// TwinCAT 3 PLC project WidgetSample
// ProgramVersion: 3.1.4026.20
// libraries:
//   Tc2_Standard, * (Beckhoff Automation GmbH)
//   Tc2_System, * (Beckhoff Automation GmbH)
//   Tc3_IotCommunicator, * (Beckhoff Automation GmbH)
//   Tc3_Module, * (Beckhoff Automation GmbH)
// project tree:
//   DUTs/4ChannelLED/ ST_Widgets_RGBWEL2564.TcDUT, ST_Widget_RGBWEL2564_Template.TcDUT
//   DUTs/AC/ ST_Widgets_AC.TcDUT, ST_Widget_AC_AlternativeTemplate.TcDUT, ST_Widget_AC_Template.TcDUT
//   DUTs/BarChart/ ST_Widgets_BarChart.TcDUT, ST_Widget_BarChart_Template.TcDUT
//   DUTs/Blinds/ ST_Widgets_Blinds.TcDUT, ST_Widget_SimpleBlinds_Template.TcDUT, ST_Widget_Blinds_Template.TcDUT
//   DUTs/ChargingStation/ ST_Widgets_ChargingStations.TcDUT, ST_Widget_ChargingStation_Template.TcDUT
//   DUTs/EnergyMonitoring/ ST_Widgets_EnergyMonitoring.TcDUT, ST_Widget_EnergyMonitoring_Template.TcDUT
//   DUTs/GeneralWidget/ ST_Widgets_GeneralWidget.TcDUT, ST_Widget_GeneralWidget_AlternativeTemplate.TcDUT, ST_Widget_GeneralWidget_Template.TcDUT
//   DUTs/Lighting/ ST_Widgets_Lightings.TcDUT, ST_Widget_Lighting_Template.TcDUT
//   DUTs/Plugs/ ST_Widgets_Plugs.TcDUT, ST_Widget_Plug_Template.TcDUT
//   DUTs/RGBW/ ST_Widgets_RGBW.TcDUT, ST_Widget_RGBW_Template.TcDUT
//   DUTs/ ST_JsonData.TcDUT, ST_WidgetData.TcDUT, ST_Widgets_Overview.TcDUT
//   DUTs/TimeSwitch/ ST_Widgets_TimeSwitch.TcDUT, ST_Widget_TimeSwitch_Template.TcDUT
//   DUTs/Ventilation/ ST_Widgets_Ventilation.TcDUT, ST_Widget_Ventilation_AlternativeTemplate.TcDUT, ST_Widget_Ventilation_Template.TcDUT
//   GVLs/ GVL_Widgets.TcGVL
//   / PlcTask.TcTTO
//   POUs/ MAIN.TcPOU, WidgetValues.TcPOU
// real-time tasks:
//   TASK PlcTask: cycle T#10ms, priority 20, ADS port 350

CONFIGURATION WidgetSample
    RESOURCE PLC ON TwinCAT3
        TASK PlcTask(INTERVAL := T#10ms, PRIORITY := 20);
        PROGRAM MAIN WITH PlcTask : MAIN;
    END_RESOURCE
END_CONFIGURATION

// ---- DUTs/4ChannelLED/ST_Widgets_RGBWEL2564.TcDUT
TYPE ST_Widgets_RGBWEL2564 :
STRUCT
	{attribute 'iot.ReadOnly' := 'true'}
	{attribute 'iot.DisplayName' := ' RGBW EL2564 Sample 1'}
	{attribute 'iot.WidgetType' := 'RGBWEL2564'}
	{attribute 'iot.LedRedSliderVisible' := 'true'}
	{attribute 'iot.LedGreenSliderVisible' := 'true'}
	{attribute 'iot.LedBlueSliderVisible' := 'true'}
	{attribute 'iot.LedWhiteSliderVisible' := 'true'}
	{attribute 'iot.LedModeVisible' := 'false'}
	{attribute 'iot.LedModeChangeable' := 'false'}
	stRGBWLed1	: ST_Widget_RGBWEL2564_Template;
	
	{attribute 'iot.ReadOnly' := 'false'}
	{attribute 'iot.DisplayName' := 'RGBW EL2564 Sample 2'}
	{attribute 'iot.WidgetType' := 'RGBWEL2564'}
	{attribute 'iot.LedRedSliderVisible' := 'true'}
	{attribute 'iot.LedGreenSliderVisible' := 'true'}
	{attribute 'iot.LedBlueSliderVisible' := 'true'}
	{attribute 'iot.LedWhiteSliderVisible' := 'true'}
	{attribute 'iot.LedModeVisible' := 'true'}
	{attribute 'iot.LedModeChangeable' := 'true'}
	stRGBWLed2	: ST_Widget_RGBWEL2564_Template;
	
	{attribute 'iot.ReadOnly' := 'false'}
	{attribute 'iot.DisplayName' := 'RGBW EL2564 Sample 3'}
	{attribute 'iot.WidgetType' := 'RGBWEL2564'}
	{attribute 'iot.LedRedSliderVisible' := 'true'}
	{attribute 'iot.LedGreenSliderVisible' := 'true'}
	{attribute 'iot.LedBlueSliderVisible' := 'true'}
	{attribute 'iot.LedWhiteSliderVisible' := 'true'}
	{attribute 'iot.LedModeVisible' := 'true'}
	{attribute 'iot.LedModeChangeable' := 'true'}
	stRGBWLed3	: ST_Widget_RGBWEL2564_Template;
END_STRUCT
END_TYPE

// ---- DUTs/4ChannelLED/ST_Widget_RGBWEL2564_Template.TcDUT
TYPE ST_Widget_RGBWEL2564_Template :
STRUCT
	sDisplayName	: STRING := ''; // Insert STRING here to overwrite iot.DisplayName

	bOn				: BOOL;
	
	nRed			: INT;
	nGreen			: INT;
	nBlue			: INT;
	nWhite			: INT;

	sMode			: STRING; // can be set to any value, does not have to match the array below
	aModes			: ARRAY[0..1] OF STRING;
END_STRUCT
END_TYPE

// ---- DUTs/AC/ST_Widgets_AC.TcDUT
TYPE ST_Widgets_AC :
STRUCT
	{attribute 'iot.ReadOnly' := 'false'}
	{attribute 'iot.DisplayName' := 'AC Sample 1'}
	{attribute 'iot.WidgetType' := 'AC'}
	{attribute 'iot.ACValueRequestVisible' := 'true'}
	{attribute 'iot.ACSliderVisible' := 'false'}
	{attribute 'iot.ACModeVisible' := 'false'}
	{attribute 'iot.ACModeChangeable' := 'false'}
	{attribute 'iot.ACModeStrengthVisible' := 'true'}
	{attribute 'iot.ACModeStrengthChangeable' := 'true'}
	{attribute 'iot.ACModeLamellaVisible' := 'true'}
	{attribute 'iot.ACModeLamellaChangeable' := 'true'}
	stAC1			: ST_Widget_AC_AlternativeTemplate;
	
	{attribute 'iot.ReadOnly' := 'false'}
	{attribute 'iot.DisplayName' := 'AC Sample 2'}
	{attribute 'iot.WidgetType' := 'AC'}
	{attribute 'iot.ACValueRequestVisible' := 'true'}
	{attribute 'iot.ACSliderVisible' := 'true'}
	{attribute 'iot.ACModeVisible' := 'true'}
	{attribute 'iot.ACModeChangeable' := 'true'}
	{attribute 'iot.ACModeStrengthVisible' := 'true'}
	{attribute 'iot.ACModeStrengthChangeable' := 'true'}
	{attribute 'iot.ACModeLamellaVisible' := 'true'}
	{attribute 'iot.ACModeLamellaChangeable' := 'true'}
	stAC2			: ST_Widget_AC_Template;
	
	{attribute 'iot.ReadOnly' := 'true'}
	{attribute 'iot.DisplayName' := 'AC Sample 3'}
	{attribute 'iot.WidgetType' := 'AC'}
	{attribute 'iot.ACValueRequestVisible' := 'false'}
	{attribute 'iot.ACSliderVisible' := 'true'}
	{attribute 'iot.ACModeVisible' := 'true'}
	{attribute 'iot.ACModeChangeable' := 'false'}
	{attribute 'iot.ACModeStrengthVisible' := 'true'}
	{attribute 'iot.ACModeStrengthChangeable' := 'false'}
	{attribute 'iot.ACModeLamellaVisible' := 'false'}
	{attribute 'iot.ACModeLamellaChangeable' := 'false'}
	stAC3			: ST_Widget_AC_Template;
END_STRUCT
END_TYPE

// ---- DUTs/AC/ST_Widget_AC_AlternativeTemplate.TcDUT
TYPE ST_Widget_AC_AlternativeTemplate :
STRUCT
	sDisplayName	: STRING := ''; // Insert STRING here to overwrite iot.DisplayName

	nAcMode			: INT;	// 0: Off, 1: Cooling, 2: Ventilating, 3: Heating, 4: Cooling Off, 5: Ventilating Off, 6: Heating Off
	
	{attribute 'iot.Unit':='°F'}
	{attribute 'iot.MinValue':='64'}
	{attribute 'iot.MaxValue':='73'}
	nTemperature		: LREAL;	
	nTemperatureRequest : LREAL;
	
	sMode			: STRING; // can be set to any value, does not have to match the array below
	aModes			: ARRAY[0..2] OF STRING;
	sMode_Strength	: STRING;
	aModes_Strength	: ARRAY[0..2] OF STRING;
	sMode_Lamella	: STRING;
	aModes_Lamella	: ARRAY[0..1] OF STRING;
END_STRUCT
END_TYPE

// ---- DUTs/AC/ST_Widget_AC_Template.TcDUT
TYPE ST_Widget_AC_Template :
STRUCT
	sDisplayName	: STRING := ''; // Insert STRING here to overwrite iot.DisplayName

	nAcMode			: INT;	// 0: Off, 1: Cooling, 2: Ventilating, 3: Heating, 4: Cooling Off, 5: Ventilating Off, 6: Heating Off
	
	{attribute 'iot.Unit':='°C'}
	{attribute 'iot.MinValue':='18'}
	{attribute 'iot.MaxValue':='23'}
	nTemperature		: LREAL;	
	nTemperatureRequest : LREAL;
	
	sMode			: STRING; // can be set to any value, does not have to match the array below
	aModes			: ARRAY[0..2] OF STRING;
	sMode_Strength	: STRING;
	aModes_Strength	: ARRAY[0..2] OF STRING;
	sMode_Lamella	: STRING;
	aModes_Lamella	: ARRAY[0..1] OF STRING;
END_STRUCT
END_TYPE

// ---- DUTs/BarChart/ST_Widgets_BarChart.TcDUT
TYPE ST_Widgets_BarChart :
STRUCT
	{attribute 'iot.DisplayName' := 'Chart Widget'}
	{attribute 'iot.WidgetType' := 'BarChart'}
	{attribute 'iot.ChartXAxisLabel' := 'Power consumption'}
	{attribute 'iot.ChartYAxisLabel' := 'Weekdays'}
	{attribute 'iot.Unit' := 'kW/h'}
	{attribute 'iot.ChartLegendVisible' := 'true'}
	{attribute 'iot.ChartValuesVisible' := 'true'}
	{attribute 'iot.MinValue':='0'}
	{attribute 'iot.MaxValue':='1550'}
	{attribute 'iot.ChartBarColor1' := '#FF80AC'}
	{attribute 'iot.ChartBarColor2' := '#FF00FF'}
	stBarChart1	: St_Widget_BarChart_Template;
	
	{attribute 'iot.DisplayName' := 'Chart Widget'}
	{attribute 'iot.WidgetType' := 'BarChart'}
	{attribute 'iot.ChartXAxisLabel' := 'Power consumption'}
	{attribute 'iot.ChartYAxisLabel' := 'Weekdays'}
	{attribute 'iot.Unit' := 'kW/h'}
	{attribute 'iot.ChartLegendVisible' := 'true'}
	{attribute 'iot.ChartValuesVisible' := 'true'}
	{attribute 'iot.MinValue':='0'}
	{attribute 'iot.MaxValue':='1600'}
	{attribute 'iot.ChartBarColor1' := '#00FFFF'}
	{attribute 'iot.ChartBarColor2' := '#0091AA'}
	stBarChart2	: St_Widget_BarChart_Template;
END_STRUCT
END_TYPE

// ---- DUTs/BarChart/ST_Widget_BarChart_Template.TcDUT
TYPE ST_Widget_BarChart_Template :
STRUCT
	sDisplayName	: STRING := '';

	aDataSeries			: ARRAY[0..6] OF INT;
	aComparismDataSeries: ARRAY[0..6] OF INT;
	aDataSeriesIdentifier:ARRAY[0..6] OF STRING;
	
	aLegendLabels		: ARRAY[0..1] OF STRING;
END_STRUCT
END_TYPE

// ---- DUTs/Blinds/ST_Widgets_Blinds.TcDUT
TYPE ST_Widgets_Blinds :
STRUCT
	{attribute 'iot.ReadOnly' := 'true'}
	{attribute 'iot.DisplayName' := 'Blinds Sample 1'}
	{attribute 'iot.WidgetType' := 'Blinds'}
	{attribute 'iot.BlindsPositionValueVisible' := 'true'}
	{attribute 'iot.BlindsPositionSliderVisible' := 'true'}
	{attribute 'iot.BlindsAngleValueVisible' := 'false'} 
	{attribute 'iot.BlindsAngleSliderVisible' := 'false'}
	{attribute 'iot.BlindsModeVisible' := 'true'} 
	{attribute 'iot.BlindsModeChangeable' := 'false'}
	stBlinds1	: ST_Widget_Blinds_Template;
	
	{attribute 'iot.ReadOnly' := 'false'}
	{attribute 'iot.DisplayName' := 'Blinds Sample 2'}
	{attribute 'iot.WidgetType' := 'Blinds'}
	{attribute 'iot.BlindsPositionValueVisible' := 'true'}
	{attribute 'iot.BlindsPositionSliderVisible' := 'true'}
	{attribute 'iot.BlindsAngleValueVisible' := 'false'} 
	{attribute 'iot.BlindsAngleSliderVisible' := 'false'}
	{attribute 'iot.BlindsModeVisible' := 'false'} 
	{attribute 'iot.BlindsModeChangeable' := 'false'}
	stBlinds2	: ST_Widget_Blinds_Template;
	
	{attribute 'iot.ReadOnly' := 'false'}
	{attribute 'iot.DisplayName' := 'Blinds Sample 3'}
	{attribute 'iot.WidgetType' := 'Blinds'}
	{attribute 'iot.BlindsPositionValueVisible' := 'true'}
	{attribute 'iot.BlindsPositionSliderVisible' := 'true'}
	{attribute 'iot.BlindsAngleValueVisible' := 'true'} 
	{attribute 'iot.BlindsAngleSliderVisible' := 'true'}
	{attribute 'iot.BlindsModeVisible' := 'true'} 
	{attribute 'iot.BlindsModeChangeable' := 'true'}
	stBlinds3	: ST_Widget_Blinds_Template;
	
	{attribute 'iot.ReadOnly' := 'false'}
	{attribute 'iot.DisplayName' := 'Simple Blinds Sample 1'}
	{attribute 'iot.WidgetType' := 'SimpleBlinds'}
	{attribute 'iot.BlindsPositionSliderVisible' := 'true'}
	stSimpleBlinds1	: ST_Widget_SimpleBlinds_Template;
	
	{attribute 'iot.ReadOnly' := 'false'}
	{attribute 'iot.DisplayName' := 'Simple Blinds Sample 2'}
	{attribute 'iot.WidgetType' := 'SimpleBlinds'}
	{attribute 'iot.BlindsPositionSliderVisible' := 'false'}
	stSimpleBlinds2	: ST_Widget_SimpleBlinds_Template;
END_STRUCT
END_TYPE

// ---- DUTs/Blinds/ST_Widget_SimpleBlinds_Template.TcDUT
TYPE ST_Widget_SimpleBlinds_Template :
STRUCT
	sDisplayName		: STRING := ''; // Insert STRING here to overwrite iot.DisplayName
	
	bPositionUp			: BOOL;
	bPositionDown		: BOOL;
	{attribute 'iot.MinValue':='0'}
	{attribute 'iot.MaxValue':='100'}
	nPositionValue		: INT;
END_STRUCT
END_TYPE

// ---- DUTs/Blinds/ST_Widget_Blinds_Template.TcDUT
TYPE ST_Widget_Blinds_Template :
STRUCT
	sDisplayName		: STRING := ''; // Insert STRING here to overwrite iot.DisplayName
	bActive				: BOOL;
	bPositionUp			: BOOL;
	bPositionDown		: BOOL;
	bAngleUp			: BOOL;
	bAngleDown			: BOOL;
	{attribute 'iot.Unit':='%'}
	{attribute 'iot.MinValue':='0'}
	{attribute 'iot.MaxValue':='100'}
	nPositionValue		: INT;	
	nPositionRequest 	: INT;
	{attribute 'iot.Unit':='°'}
	{attribute 'iot.MinValue':='-90'}
	{attribute 'iot.MaxValue':='90'}
	nAngleValue			: INT;
	nAngleRequest 		: INT;	
	sMode				: STRING; // can be set to any value, does not have to match the array below
	aModes				: ARRAY[0..1] OF STRING;
END_STRUCT
END_TYPE

// ---- DUTs/ChargingStation/ST_Widgets_ChargingStations.TcDUT
TYPE ST_Widgets_ChargingStations :
STRUCT
	{attribute 'iot.ReadOnly' := 'false'}
	{attribute 'iot.DisplayName' := 'Charging Station Sample 1'}
	{attribute 'iot.WidgetType' := 'ChargingStation'}
	{attribute 'iot.ChargingStationReserveVisible' := 'true'} 
	{attribute 'iot.ChargingStationPhase2Visible' := 'true'} 
	{attribute 'iot.ChargingStationPhase3Visible' := 'true'} 
	stChargingStation1	: ST_Widget_ChargingStation_Template;
	
	{attribute 'iot.ReadOnly' := 'false'}
	{attribute 'iot.DisplayName' := 'Charging Station Sample 2'}
	{attribute 'iot.WidgetType' := 'ChargingStation'}
	{attribute 'iot.ChargingStationReserveVisible' := 'false'} 
	{attribute 'iot.ChargingStationPhase2Visible' := 'true'} 
	{attribute 'iot.ChargingStationPhase3Visible' := 'false'} 
	stChargingStation2	: ST_Widget_ChargingStation_Template;
END_STRUCT
END_TYPE

// ---- DUTs/ChargingStation/ST_Widget_ChargingStation_Template.TcDUT
TYPE ST_Widget_ChargingStation_Template :
STRUCT
	sDisplayName				: STRING;
	
	bStartCharging				: BOOL;
	bStopCharging				: BOOL;
	bReserveCharging			: BOOL;
	
	sStatus						: STRING;	
	nBatteryLevel				: UINT;
	nCurrentPower				: LREAL;
	aThreePhaseMaxPower			: ARRAY[0..2] OF LREAL;
	aThreePhaseCurrentPower		: ARRAY[0..2] OF LREAL;
	aThreePhaseAmperage			: ARRAY[0..2] OF LREAL;
	aThreePhaseVoltage			: ARRAY[0..2] OF LREAL;
	nChargingTime				: UDINT;
	nChargingEnergy				: LREAL;
END_STRUCT
END_TYPE

// ---- DUTs/EnergyMonitoring/ST_Widgets_EnergyMonitoring.TcDUT
TYPE ST_Widgets_EnergyMonitoring :
STRUCT
	{attribute 'iot.ReadOnly' := 'false'}
	{attribute 'iot.DisplayName' := 'Energy Monitoring Sample 1'}
	{attribute 'iot.WidgetType' := 'EnergyMonitoring'}
	{attribute 'iot.EnergyMonitoringPhase2Visible' := 'true'} 
	{attribute 'iot.EnergyMonitoringPhase3Visible' := 'true'} 
	stEnergyMonitoring1	: ST_Widget_EnergyMonitoring_Template;
	
	{attribute 'iot.ReadOnly' := 'false'}
	{attribute 'iot.DisplayName' := 'Energy Monitoring Sample 2'}
	{attribute 'iot.WidgetType' := 'EnergyMonitoring'}
	{attribute 'iot.EnergyMonitoringPhase2Visible' := 'true'} 
	{attribute 'iot.EnergyMonitoringPhase3Visible' := 'false'} 
	stEnergyMonitoring2	: ST_Widget_EnergyMonitoring_Template;
	
	{attribute 'iot.ReadOnly' := 'false'}
	{attribute 'iot.DisplayName' := 'Energy Monitoring Sample 3'}
	{attribute 'iot.WidgetType' := 'EnergyMonitoring'}
	{attribute 'iot.EnergyMonitoringPhase2Visible' := 'false'} 
	{attribute 'iot.EnergyMonitoringPhase3Visible' := 'false'} 
	stEnergyMonitoring3	: ST_Widget_EnergyMonitoring_Template;
END_STRUCT
END_TYPE

// ---- DUTs/EnergyMonitoring/ST_Widget_EnergyMonitoring_Template.TcDUT
TYPE ST_Widget_EnergyMonitoring_Template :
STRUCT
	sDisplayName				: STRING;
	
	sStatus						: STRING;	
	aThreePhaseMaxPower			: ARRAY[0..2] OF LREAL;
	aThreePhaseCurrentPower		: ARRAY[0..2] OF LREAL;
	aThreePhasePowerUnits		: ARRAY[0..2] OF STRING;
	aThreePhaseAmperage			: ARRAY[0..2] OF LREAL;
	aThreePhaseAmperageUnits	: ARRAY[0..2] OF STRING;
	aThreePhaseVoltage			: ARRAY[0..2] OF LREAL;
	aThreePhaseVoltageUnits		: ARRAY[0..2] OF STRING;
	nPowerQualityFactor			: LREAL;	
	nCurrentPower				: LREAL;
	sPowerUnit					: STRING;
	nEnergy						: LREAL;
	sEnergyUnit					: STRING;
END_STRUCT
END_TYPE

// ---- DUTs/GeneralWidget/ST_Widgets_GeneralWidget.TcDUT
TYPE ST_Widgets_GeneralWidget :
STRUCT
	{attribute 'iot.ReadOnly' := 'true'}
	{attribute 'iot.DisplayName' := 'General Widget Sample 1'}
	{attribute 'iot.WidgetType' := 'General'}
	{attribute 'iot.GeneralWidgetIcon' := 'Snowflake_Blue'}
	{attribute 'iot.GeneralWidgetColor' := '#FFDCDCDC'}
	{attribute 'iot.GeneralValue1SwitchVisible' := 'true'}
	{attribute 'iot.GeneralValue2Visible' := 'false'}
	{attribute 'iot.GeneralValue2SliderVisible' := 'false'}
	{attribute 'iot.GeneralValue2SliderValuesVisible' := 'false'}
	{attribute 'iot.GeneralValue2SliderButtonsVisible' := 'false'}
	{attribute 'iot.GeneralValue2SliderButtonsInverted' := 'false'}
	{attribute 'iot.GeneralValue3Visible' := 'false'} 
	{attribute 'iot.GeneralValue3SliderVisible' := 'false'}
	{attribute 'iot.GeneralValue3SliderValuesVisible' := 'false'}
	{attribute 'iot.GeneralValue3SliderButtonsVisible' := 'false'}
	{attribute 'iot.GeneralValue3SliderButtonsInverted' := 'false'}
	{attribute 'iot.GeneralMode1Visible' := 'true'} 
	{attribute 'iot.GeneralMode1Changeable' := 'false'}
	{attribute 'iot.GeneralMode2Visible' := 'false'} 
	{attribute 'iot.GeneralMode2Changeable' := 'false'}
	{attribute 'iot.GeneralMode3Visible' := 'false'} 
	{attribute 'iot.GeneralMode3Changeable' := 'false'}
	stGeneral1	: ST_Widget_GeneralWidget_Template;
	
	{attribute 'iot.ReadOnly' := 'false'}
	{attribute 'iot.DisplayName' := 'General Widget Sample 2'}
	{attribute 'iot.WidgetType' := 'General'}
	{attribute 'iot.GeneralWidgetIcon' := 'Co2'}
	{attribute 'iot.GeneralWidgetColor' := '#66FF0000'}
	{attribute 'iot.GeneralValue1SwitchVisible' := 'true'}
	{attribute 'iot.GeneralValue2Visible' := 'true'}
	{attribute 'iot.GeneralValue2SliderVisible' := 'true'}
	{attribute 'iot.GeneralValue2SliderValuesVisible' := 'true'}
	{attribute 'iot.GeneralValue2SliderButtonsVisible' := 'true'}
	{attribute 'iot.GeneralValue2SliderButtonsInverted' := 'true'}
	{attribute 'iot.GeneralValue3Visible' := 'false'} 
	{attribute 'iot.GeneralValue3SliderVisible' := 'false'}
	{attribute 'iot.GeneralValue3SliderValuesVisible' := 'false'}
	{attribute 'iot.GeneralValue3SliderButtonsVisible' := 'false'}
	{attribute 'iot.GeneralValue3SliderButtonsInverted' := 'false'}
	{attribute 'iot.GeneralMode1Visible' := 'true'} 
	{attribute 'iot.GeneralMode1Changeable' := 'true'}
	{attribute 'iot.GeneralMode2Visible' := 'true'} 
	{attribute 'iot.GeneralMode2Changeable' := 'false'}
	{attribute 'iot.GeneralMode3Visible' := 'false'} 
	{attribute 'iot.GeneralMode3Changeable' := 'false'}
	stGeneral2	: ST_Widget_GeneralWidget_Template;
	
	{attribute 'iot.ReadOnly' := 'false'}
	{attribute 'iot.DisplayName' := 'General Widget Sample 3'}
	{attribute 'iot.WidgetType' := 'General'}
	{attribute 'iot.GeneralWidgetIcon' := 'Room'}
	{attribute 'iot.GeneralWidgetColor' := '#FF2F4F4F'}
	{attribute 'iot.GeneralValue1SwitchVisible' := 'true'}
	{attribute 'iot.GeneralValue2Visible' := 'true'}
	{attribute 'iot.GeneralValue2SliderVisible' := 'true'}
	{attribute 'iot.GeneralValue2SliderValuesVisible' := 'true'}
	{attribute 'iot.GeneralValue2SliderButtonsVisible' := 'true'}
	{attribute 'iot.GeneralValue2SliderButtonsInverted' := 'true'}
	{attribute 'iot.GeneralValue3Visible' := 'true'} 
	{attribute 'iot.GeneralValue3SliderVisible' := 'true'}
	{attribute 'iot.GeneralValue3SliderValuesVisible' := 'true'}
	{attribute 'iot.GeneralValue3SliderButtonsVisible' := 'true'}
	{attribute 'iot.GeneralValue3SliderButtonsInverted' := 'false'}
	{attribute 'iot.GeneralMode1Visible' := 'true'} 
	{attribute 'iot.GeneralMode1Changeable' := 'true'}
	{attribute 'iot.GeneralMode2Visible' := 'true'} 
	{attribute 'iot.GeneralMode2Changeable' := 'true'}
	{attribute 'iot.GeneralMode3Visible' := 'true'} 
	{attribute 'iot.GeneralMode3Changeable' := 'true'}
	stGeneral3	: ST_Widget_GeneralWidget_AlternativeTemplate;
END_STRUCT
END_TYPE

// ---- DUTs/GeneralWidget/ST_Widget_GeneralWidget_AlternativeTemplate.TcDUT
TYPE ST_Widget_GeneralWidget_AlternativeTemplate :
STRUCT
	sDisplayName	: STRING := ''; // Insert STRING here to overwrite iot.DisplayName

	bValue1			: BOOL;
	
	{attribute 'iot.Unit':='$$'}
	{attribute 'iot.MinValue':='0'}
	{attribute 'iot.MaxValue':='365'}
	nValue2			: INT;	
	nValue2Request 	: INT;
	bValue2Up		: BOOL;
	bValue2Down		: BOOL;
	
	{attribute 'iot.Unit':='€'}
	{attribute 'iot.MinValue':='0'}
	{attribute 'iot.MaxValue':='1000'}
	nValue3			: INT;
	nValue3Request 	: INT;
	bValue3Up		: BOOL;
	bValue3Down		: BOOL;
	
	sMode1			: STRING; // can be set to any value, does not have to match the array below
	aModes1			: ARRAY[0..3] OF STRING;
	sMode2			: STRING;
	aModes2			: ARRAY[0..2] OF STRING;
	sMode3			: STRING;
	aModes3			: ARRAY[0..1] OF STRING;
END_STRUCT
END_TYPE

// ---- DUTs/GeneralWidget/ST_Widget_GeneralWidget_Template.TcDUT
TYPE ST_Widget_GeneralWidget_Template :
STRUCT
	sDisplayName	: STRING := ''; // Insert STRING here to overwrite iot.DisplayName

	bValue1			: BOOL;
	
	{attribute 'iot.Unit':='%'}
	{attribute 'iot.MinValue':='0'}
	{attribute 'iot.MaxValue':='100'}
	nValue2			: INT;	
	nValue2Request 	: INT;
	bValue2Up		: BOOL;
	bValue2Down		: BOOL;
	
	{attribute 'iot.Unit':='°'}
	{attribute 'iot.MinValue':='-90'}
	{attribute 'iot.MaxValue':='90'}
	nValue3			: INT;
	nValue3Request 	: INT;
	bValue3Up		: BOOL;
	bValue3Down		: BOOL;
	
	sMode1			: STRING; // can be set to any value, does not have to match the array below
	aModes1			: ARRAY[0..1] OF STRING;
	sMode2			: STRING;
	aModes2			: ARRAY[0..2] OF STRING;
	sMode3			: STRING;
	aModes3			: ARRAY[0..1] OF STRING;
END_STRUCT
END_TYPE

// ---- DUTs/Lighting/ST_Widgets_Lightings.TcDUT
TYPE ST_Widgets_Lightings :
STRUCT
	{attribute 'iot.ReadOnly' := 'true'}
	{attribute 'iot.DisplayName' := 'Lighting Sample 1'}
	{attribute 'iot.WidgetType' := 'Lighting'}
	{attribute 'iot.LightValueVisible' := 'false'}
	{attribute 'iot.LightSliderVisible' := 'false'}
	{attribute 'iot.LightModeVisible' := 'false'}
	{attribute 'iot.LightModeChangeable' := 'false'}
	stLighting1	: ST_Widget_Lighting_Template;
	
	{attribute 'iot.ReadOnly' := 'false'}
	{attribute 'iot.DisplayName' := 'Lighting Sample 2'}
	{attribute 'iot.WidgetType' := 'Lighting'}
	{attribute 'iot.LightValueVisible' := 'false'}
	{attribute 'iot.LightSliderVisible' := 'true'}
	{attribute 'iot.LightModeVisible' := 'true'}
	{attribute 'iot.LightModeChangeable' := 'true'}
	stLighting2	: ST_Widget_Lighting_Template;
	
	{attribute 'iot.ReadOnly' := 'false'}
	{attribute 'iot.DisplayName' := 'Lighting Sample 3'}
	{attribute 'iot.WidgetType' := 'Lighting'}
	{attribute 'iot.LightValueVisible' := 'true'}
	{attribute 'iot.LightSliderVisible' := 'true'}
	{attribute 'iot.LightModeVisible' := 'true'}
	{attribute 'iot.LightModeChangeable' := 'true'}
	stLighting3	: ST_Widget_Lighting_Template;
END_STRUCT
END_TYPE

// ---- DUTs/Lighting/ST_Widget_Lighting_Template.TcDUT
TYPE ST_Widget_Lighting_Template :
STRUCT
	bLight		: BOOL;
	{attribute 'iot.Unit':='%'}
	{attribute 'iot.MinValue':='0'}
	{attribute 'iot.MaxValue':='100'}
	nLight		: INT;	
	sMode		: STRING ;
	aModes		: ARRAY[0..1] OF STRING;
END_STRUCT
END_TYPE

// ---- DUTs/Plugs/ST_Widgets_Plugs.TcDUT
TYPE ST_Widgets_Plugs :
STRUCT
	{attribute 'iot.ReadOnly' := 'false'}
	{attribute 'iot.DisplayName' := 'Plug Sample 1'}
	{attribute 'iot.WidgetType' := 'Plug'}
	{attribute 'iot.PlugModeVisible' := 'false'}
	{attribute 'iot.PlugModeChangeable' := 'false'}
	stPlug1		: ST_Widget_Plug_Template;
	
	{attribute 'iot.ReadOnly' := 'false'}
	{attribute 'iot.DisplayName' := 'Plug Sample 2'}
	{attribute 'iot.WidgetType' := 'Plug'}
	{attribute 'iot.PlugModeVisible' := 'true'}
	{attribute 'iot.PlugModeChangeable' := 'true'}
	stPlug2		: ST_Widget_Plug_Template;
END_STRUCT
END_TYPE

// ---- DUTs/Plugs/ST_Widget_Plug_Template.TcDUT
TYPE ST_Widget_Plug_Template :
STRUCT
	sDisplayName	: STRING := ''; // Insert STRING here to overwrite iot.DisplayName

	bOn				: BOOL;

	sMode			: STRING; // can be set to any value, does not have to match the array below
	aModes			: ARRAY[0..1] OF STRING;
END_STRUCT
END_TYPE

// ---- DUTs/RGBW/ST_Widgets_RGBW.TcDUT
TYPE ST_Widgets_RGBW :
STRUCT
	{attribute 'iot.ReadOnly' := 'true'}
	{attribute 'iot.DisplayName' := 'RGBW Lighting Sample 1'}
	{attribute 'iot.WidgetType' := 'RGBW'}
	{attribute 'iot.LightValueVisible' := 'false'}
	{attribute 'iot.LightSliderVisible' := 'false'}
	{attribute 'iot.LightColorPaletteVisible' := 'true'}
	{attribute 'iot.LightColorTemperatureSliderVisible' := 'true'}
	{attribute 'iot.LightWhiteSliderVisible' := 'false'}
	{attribute 'iot.LightModeVisible' := 'false'}
	{attribute 'iot.LightModeChangeable' := 'false'}
	stRGB1	: ST_Widget_RGBW_Template;
	
	{attribute 'iot.ReadOnly' := 'false'}
	{attribute 'iot.DisplayName' := 'RGBW Lighting Sample 2'}
	{attribute 'iot.WidgetType' := 'RGBW'}
	{attribute 'iot.LightValueVisible' := 'true'}
	{attribute 'iot.LightSliderVisible' := 'true'}
	{attribute 'iot.LightColorPaletteVisible' := 'true'}
	{attribute 'iot.LightColorTemperatureSliderVisible' := 'false'}
	{attribute 'iot.LightWhiteSliderVisible' := 'false'}
	{attribute 'iot.LightModeVisible' := 'true'}
	{attribute 'iot.LightModeChangeable' := 'true'}
	stRGB2	: ST_Widget_RGBW_Template;
	
	{attribute 'iot.ReadOnly' := 'false'}
	{attribute 'iot.DisplayName' := 'RGBW Lighting Sample 3'}
	{attribute 'iot.WidgetType' := 'RGBW'}
	{attribute 'iot.LightValueVisible' := 'true'}
	{attribute 'iot.LightSliderVisible' := 'true'}
	{attribute 'iot.LightColorPaletteVisible' := 'true'}
	{attribute 'iot.LightColorTemperatureSliderVisible' := 'true'}
	{attribute 'iot.LightWhiteSliderVisible' := 'true'}
	{attribute 'iot.LightModeVisible' := 'true'}
	{attribute 'iot.LightModeChangeable' := 'true'}
	stRGB3	: ST_Widget_RGBW_Template;
END_STRUCT
END_TYPE

// ---- DUTs/RGBW/ST_Widget_RGBW_Template.TcDUT
TYPE ST_Widget_RGBW_Template :
STRUCT
	sDisplayName	: STRING := '';

	bLight		: BOOL;
	{attribute 'iot.Unit':='%'}
	{attribute 'iot.MinValue':='0'}
	{attribute 'iot.MaxValue':='100'}
	nLight		: INT;	
	
	// Attention: If using OnChange mechanism, HueValue & Saturation have to be send together
	// 			  even if only one of them is changed
	nHueValue	: INT;
	nSaturation	: INT;
	
	{attribute 'iot.MinValue':='2400'}
	{attribute 'iot.MaxValue':='6500'}
	nColorTemperature : INT;
	nWhite : INT;
	
	sMode		: STRING;
	aModes		: ARRAY[0..1] OF STRING;
END_STRUCT
END_TYPE

// ---- DUTs/ST_JsonData.TcDUT
TYPE ST_JsonData :
STRUCT
	sJsonStringToSend : STRING(1000);
END_STRUCT
END_TYPE

// ---- DUTs/ST_WidgetData.TcDUT
TYPE ST_WidgetData :
STRUCT
	{attribute 'iot.NestedStructIcon' := 'Floor'}
	{attribute 'iot.DisplayName' := 'All Widgets Overview'}
	stWidgetsOverview	: ST_Widgets_Overview;
	
	{attribute 'iot.NestedStructIcon' := 'Lightbulb'}
	{attribute 'iot.DisplayName' := 'Light Widgets'}
	stLights			: ST_Widgets_Lightings;
	
	{attribute 'iot.NestedStructIcon' := 'Lightbulb'}
	{attribute 'iot.DisplayName' := 'RGBW Widgets'}
	stRGBW				: ST_Widgets_RGBW;
	
	{attribute 'iot.NestedStructIcon' := 'Lightbulb'}
	{attribute 'iot.DisplayName' := 'RGBW EL2564 Widgets'}
	stRGBWEL2564		: ST_Widgets_RGBWEL2564;
	
	{attribute 'iot.NestedStructIcon' := 'Blinds'}
	{attribute 'iot.DisplayName' := 'Blinds Widgets'}
	stBlinds			: ST_Widgets_Blinds;
	
	{attribute 'iot.NestedStructIcon' := 'Plug'}
	{attribute 'iot.DisplayName' := 'Plug Widgets'}
	stPlugs				: ST_Widgets_Plugs;
	
	{attribute 'iot.NestedStructIcon' := 'Temperature'}
	{attribute 'iot.DisplayName' := 'AC Widgets'}
	stAC				: ST_Widgets_AC;
	
	{attribute 'iot.NestedStructIcon' := 'Co2'}
	{attribute 'iot.DisplayName' := 'Ventilation Widgets'}
	stVentilation		: ST_Widgets_Ventilation;
	
	{attribute 'iot.NestedStructIcon' := 'Clock'}
	{attribute 'iot.DisplayName' := 'Time Switch Widgets'}
	stTimeSwitch		: ST_Widgets_TimeSwitch;
	
	{attribute 'iot.NestedStructIcon' := 'Floor'}
	{attribute 'iot.DisplayName' := 'BarChart Widgets'}
	stBarChart			: ST_Widgets_BarChart;
	
	{attribute 'iot.NestedStructIcon' := 'Charging_Station'}
	{attribute 'iot.DisplayName' := 'Charging Station Widgets'}
	stChargingStation	: ST_Widgets_ChargingStations;
	
	{attribute 'iot.NestedStructIcon' := 'Lightning'}
	{attribute 'iot.DisplayName' := 'Energy Monitoring Widgets'}
	stEnergyMonitoring	: ST_Widgets_EnergyMonitoring;
	
	{attribute 'iot.NestedStructIcon' := 'Room'}
	{attribute 'iot.DisplayName' := 'General Widgets'}
	stGeneral			: ST_Widgets_GeneralWidget;
END_STRUCT
END_TYPE

// ---- DUTs/ST_Widgets_Overview.TcDUT
TYPE ST_Widgets_Overview :
STRUCT
	{attribute 'iot.ReadOnly' := 'false'}
	{attribute 'iot.DisplayName' := 'Full-Featured Lighting'}
	{attribute 'iot.WidgetType' := 'Lighting'}
	{attribute 'iot.LightValueVisible' := 'true'}
	{attribute 'iot.LightSliderVisible' := 'true'}
	{attribute 'iot.LightModeVisible' := 'true'}
	{attribute 'iot.LightModeChangeable' := 'true'}
	stLighting		: ST_Widget_Lighting_Template;
	
	{attribute 'iot.ReadOnly' := 'false'}
	{attribute 'iot.DisplayName' := 'Full-Featured RGBW'}
	{attribute 'iot.WidgetType' := 'RGBW'}
	{attribute 'iot.LightValueVisible' := 'true'}
	{attribute 'iot.LightSliderVisible' := 'true'}
	{attribute 'iot.LightColorPaletteVisible' := 'true'}
	{attribute 'iot.LightColorTemperatureSliderVisible' := 'true'}
	{attribute 'iot.LightWhiteSliderVisible' := 'true'}
	{attribute 'iot.LightModeVisible' := 'true'}
	{attribute 'iot.LightModeChangeable' := 'true'}
	stRGBW			: ST_Widget_RGBW_Template;
	
	{attribute 'iot.ReadOnly' := 'false'}
	{attribute 'iot.DisplayName' := 'Full-Featured RGBW EL2564'}
	{attribute 'iot.WidgetType' := 'RGBWEL2564'}
	{attribute 'iot.LedRedSliderVisible' := 'true'}
	{attribute 'iot.LedGreenSliderVisible' := 'true'}
	{attribute 'iot.LedBlueSliderVisible' := 'true'}
	{attribute 'iot.LedWhiteSliderVisible' := 'true'}
	{attribute 'iot.LedModeVisible' := 'true'}
	{attribute 'iot.LedModeChangeable' := 'true'}
	stRGBWLed		: ST_Widget_RGBWEL2564_Template;
	
	{attribute 'iot.ReadOnly' := 'false'}
	{attribute 'iot.DisplayName' := 'Full-Featured Blinds'}
	{attribute 'iot.WidgetType' := 'Blinds'}
	{attribute 'iot.BlindsPositionValueVisible' := 'true'}
	{attribute 'iot.BlindsPositionSliderVisible' := 'true'}
	{attribute 'iot.BlindsAngleValueVisible' := 'true'} 
	{attribute 'iot.BlindsAngleSliderVisible' := 'true'}
	{attribute 'iot.BlindsModeVisible' := 'true'} 
	{attribute 'iot.BlindsModeChangeable' := 'true'}
	stBlinds		: ST_Widget_Blinds_Template;
	
	{attribute 'iot.ReadOnly' := 'false'}
	{attribute 'iot.DisplayName' := 'Full-Featured Simple Blinds'}
	{attribute 'iot.WidgetType' := 'SimpleBlinds'}
	{attribute 'iot.BlindsPositionSliderVisible' := 'true'}
	stSimpleBlinds	: ST_Widget_SimpleBlinds_Template;
	
	{attribute 'iot.ReadOnly' := 'false'}
	{attribute 'iot.DisplayName' := 'Full-Featured Plug'}
	{attribute 'iot.WidgetType' := 'Plug'}
	{attribute 'iot.PlugModeVisible' := 'true'}
	{attribute 'iot.PlugModeChangeable' := 'true'}
	stPlug			: ST_Widget_Plug_Template;
	
	{attribute 'iot.ReadOnly' := 'false'}
	{attribute 'iot.DisplayName' := 'Full-Featured AC'}
	{attribute 'iot.WidgetType' := 'AC'}
	{attribute 'iot.ACValueRequestVisible' := 'true'}
	{attribute 'iot.ACSliderVisible' := 'true'}
	{attribute 'iot.ACModeVisible' := 'true'}
	{attribute 'iot.ACModeChangeable' := 'true'}
	{attribute 'iot.ACModeStrengthVisible' := 'true'}
	{attribute 'iot.ACModeStrengthChangeable' := 'true'}
	{attribute 'iot.ACModeLamellaVisible' := 'true'}
	{attribute 'iot.ACModeLamellaChangeable' := 'true'}
	stAC			: ST_Widget_AC_Template;
	
	{attribute 'iot.ReadOnly' := 'false'}
	{attribute 'iot.DisplayName' := 'Full-Featured Ventilation'}
	{attribute 'iot.WidgetType' := 'Ventilation'}
	{attribute 'iot.VentilationValueRequestVisible' := 'true'}
	{attribute 'iot.VentilationSliderVisible' := 'true'}
	{attribute 'iot.VentilationModeVisible' := 'true'}
	{attribute 'iot.VentilationModeChangeable' := 'true'}
	stVentilation		: ST_Widget_Ventilation_Template;
	
	{attribute 'iot.ReadOnly' := 'false'}
	{attribute 'iot.DisplayName' := 'Full-Featured Time Switch'}
	{attribute 'iot.WidgetType' := 'TimeSwitch'}
	{attribute 'iot.TimeSwitchStartTimeVisible' := 'true'}
	{attribute 'iot.TimeSwitchEndTimeVisible' := 'true'}
	{attribute 'iot.TimeSwitchStartDateVisible' := 'true'}
	{attribute 'iot.TimeSwitchEndDateVisible' := 'true'}
	{attribute 'iot.TimeSwitchDaysVisible' := 'true'}
	{attribute 'iot.TimeSwitchModeVisible' := 'true'}
	{attribute 'iot.TimeSwitchModeChangeable' := 'true'}
	stTimeSwitch		: ST_Widget_TimeSwitch_Template;
	
	{attribute 'iot.DisplayName' := 'Full-Featured BarChart'}
	{attribute 'iot.WidgetType' := 'BarChart'}
	{attribute 'iot.ChartXAxisLabel' := 'Power consumption'}
	{attribute 'iot.ChartYAxisLabel' := 'Weekdays'}
	{attribute 'iot.Unit' := 'kW/h'}
	{attribute 'iot.ChartLegendVisible' := 'true'}
	{attribute 'iot.ChartValuesVisible' := 'true'}
	{attribute 'iot.MinValue':='0'}
	{attribute 'iot.MaxValue':='1550'}
	{attribute 'iot.ChartBarColor1' := '#00FFFF'}
	{attribute 'iot.ChartBarColor2' := '#FF00FF'}
	stBarChart			: St_Widget_BarChart_Template;
	
	{attribute 'iot.ReadOnly' := 'false'}
	{attribute 'iot.DisplayName' := 'Full-Featured Charging Station'}
	{attribute 'iot.WidgetType' := 'ChargingStation'}
	{attribute 'iot.ChargingStationReserveVisible' := 'true'} 
	{attribute 'iot.ChargingStationPhase2Visible' := 'true'} 
	{attribute 'iot.ChargingStationPhase3Visible' := 'true'} 
	stChargingStation	: ST_Widget_ChargingStation_Template;
	
	{attribute 'iot.ReadOnly' := 'false'}
	{attribute 'iot.DisplayName' := 'Full-Featured Energy Monitoring'}
	{attribute 'iot.WidgetType' := 'EnergyMonitoring'}
	{attribute 'iot.EnergyMonitoringPhase2Visible' := 'true'} 
	{attribute 'iot.EnergyMonitoringPhase3Visible' := 'true'} 
	stEnergyMonitoring	: ST_Widget_EnergyMonitoring_Template;
	
	{attribute 'iot.ReadOnly' := 'false'}
	{attribute 'iot.DisplayName' := 'Full-Featured General Widget'}
	{attribute 'iot.WidgetType' := 'General'}
	{attribute 'iot.GeneralWidgetIcon' := 'Room'}
	{attribute 'iot.GeneralWidgetColor' := '#FFFF00FF'}
	{attribute 'iot.GeneralValue1SwitchVisible' := 'true'}
	{attribute 'iot.GeneralValue2Visible' := 'true'}
	{attribute 'iot.GeneralValue2SliderVisible' := 'true'}
	{attribute 'iot.GeneralValue2SliderValuesVisible' := 'true'}
	{attribute 'iot.GeneralValue2SliderButtonsVisible' := 'true'}
	{attribute 'iot.GeneralValue2SliderButtonsInverted' := 'true'}
	{attribute 'iot.GeneralValue3Visible' := 'true'} 
	{attribute 'iot.GeneralValue3SliderVisible' := 'true'}
	{attribute 'iot.GeneralValue3SliderValuesVisible' := 'true'}
	{attribute 'iot.GeneralValue3SliderButtonsVisible' := 'true'}
	{attribute 'iot.GeneralValue3SliderButtonsInverted' := 'false'}
	{attribute 'iot.GeneralMode1Visible' := 'true'} 
	{attribute 'iot.GeneralMode1Changeable' := 'true'}
	{attribute 'iot.GeneralMode2Visible' := 'true'} 
	{attribute 'iot.GeneralMode2Changeable' := 'true'}
	{attribute 'iot.GeneralMode3Visible' := 'true'} 
	{attribute 'iot.GeneralMode3Changeable' := 'true'}
	stGeneral		: ST_Widget_GeneralWidget_Template;
END_STRUCT
END_TYPE

// ---- DUTs/TimeSwitch/ST_Widgets_TimeSwitch.TcDUT
TYPE ST_Widgets_TimeSwitch :
STRUCT
	{attribute 'iot.ReadOnly' := 'false'}
	{attribute 'iot.DisplayName' := 'Time Switch Sample 1'}
	{attribute 'iot.WidgetType' := 'TimeSwitch'}
	{attribute 'iot.TimeSwitchStartTimeVisible' := 'true'}
	{attribute 'iot.TimeSwitchEndTimeVisible' := 'true'}
	{attribute 'iot.TimeSwitchStartDateVisible' := 'true'}
	{attribute 'iot.TimeSwitchEndDateVisible' := 'true'}
	{attribute 'iot.TimeSwitchDaysVisible' := 'false'}
	{attribute 'iot.TimeSwitchModeVisible' := 'true'}
	{attribute 'iot.TimeSwitchModeChangeable' := 'false'}
	stTimeSwitch1		: ST_Widget_TimeSwitch_Template;
	
	{attribute 'iot.ReadOnly' := 'false'}
	{attribute 'iot.DisplayName' := 'Time Switch Sample 2'}
	{attribute 'iot.WidgetType' := 'TimeSwitch'}
	{attribute 'iot.TimeSwitchStartTimeVisible' := 'true'}
	{attribute 'iot.TimeSwitchEndTimeVisible' := 'true'}
	{attribute 'iot.TimeSwitchStartDateVisible' := 'false'}
	{attribute 'iot.TimeSwitchEndDateVisible' := 'false'}
	{attribute 'iot.TimeSwitchDaysVisible' := 'true'}
	{attribute 'iot.TimeSwitchModeVisible' := 'false'}
	{attribute 'iot.TimeSwitchModeChangeable' := 'false'}
	stTimeSwitch2		: ST_Widget_TimeSwitch_Template;
	
	{attribute 'iot.ReadOnly' := 'false'}
	{attribute 'iot.DisplayName' := 'Time Switch Sample 3'}
	{attribute 'iot.WidgetType' := 'TimeSwitch'}
	{attribute 'iot.TimeSwitchStartTimeVisible' := 'true'}
	{attribute 'iot.TimeSwitchEndTimeVisible' := 'true'}
	{attribute 'iot.TimeSwitchStartDateVisible' := 'true'}
	{attribute 'iot.TimeSwitchEndDateVisible' := 'true'}
	{attribute 'iot.TimeSwitchDaysVisible' := 'true'}
	{attribute 'iot.TimeSwitchModeVisible' := 'true'}
	{attribute 'iot.TimeSwitchModeChangeable' := 'true'}
	stTimeSwitch3		: ST_Widget_TimeSwitch_Template;
END_STRUCT
END_TYPE

// ---- DUTs/TimeSwitch/ST_Widget_TimeSwitch_Template.TcDUT
TYPE ST_Widget_TimeSwitch_Template :
STRUCT
	sDisplayName	: STRING := ''; // Insert STRING here to overwrite iot.DisplayName
	
	bOn				: BOOL;
	
	tStartTime		: TIME_OF_DAY;
	tEndTime		: TIME_OF_DAY;
	dStartDate		: DATE;
	dEndDate		: DATE;
	bYearly			: BOOL;
	
	bMonday			: BOOL;
	bTuesday		: BOOL;
	bWednesday		: BOOL;
	bThursday		: BOOL;
	bFriday			: BOOL;
	bSaturday		: BOOL;
	bSunday			: BOOL;
	
	sMode			: STRING; // can be set to any value, does not have to match the array below
	aModes			: ARRAY[0..1] OF STRING;
END_STRUCT
END_TYPE

// ---- DUTs/Ventilation/ST_Widgets_Ventilation.TcDUT
TYPE ST_Widgets_Ventilation :
STRUCT
	{attribute 'iot.ReadOnly' := 'true'}
	{attribute 'iot.DisplayName' := 'Ventilation Sample 1'}
	{attribute 'iot.WidgetType' := 'Ventilation'}
	{attribute 'iot.VentilationValueRequestVisible' := 'true'}
	{attribute 'iot.VentilationSliderVisible' := 'false'}
	{attribute 'iot.VentilationModeVisible' := 'false'}
	{attribute 'iot.VentilationModeChangeable' := 'false'}
	stVentilation1		: ST_Widget_Ventilation_Template;
	
	{attribute 'iot.ReadOnly' := 'false'}
	{attribute 'iot.DisplayName' := 'Ventilation Sample 2'}
	{attribute 'iot.WidgetType' := 'Ventilation'}
	{attribute 'iot.VentilationValueRequestVisible' := 'true'}
	{attribute 'iot.VentilationSliderVisible' := 'true'}
	{attribute 'iot.VentilationModeVisible' := 'true'}
	{attribute 'iot.VentilationModeChangeable' := 'false'}
	stVentilation2		: ST_Widget_Ventilation_AlternativeTemplate;
	
	{attribute 'iot.ReadOnly' := 'false'}
	{attribute 'iot.DisplayName' := 'Ventilation Sample 3'}
	{attribute 'iot.WidgetType' := 'Ventilation'}
	{attribute 'iot.VentilationValueRequestVisible' := 'true'}
	{attribute 'iot.VentilationSliderVisible' := 'true'}
	{attribute 'iot.VentilationModeVisible' := 'true'}
	{attribute 'iot.VentilationModeChangeable' := 'true'}
	stVentilation3		: ST_Widget_Ventilation_Template;
END_STRUCT
END_TYPE

// ---- DUTs/Ventilation/ST_Widget_Ventilation_AlternativeTemplate.TcDUT
TYPE ST_Widget_Ventilation_AlternativeTemplate :
STRUCT
	sDisplayName	: STRING := ''; // Insert STRING here to overwrite iot.DisplayName

	bOn				: BOOL;
	
	{attribute 'iot.Unit':='ppm'}
	{attribute 'iot.MinValue':='600'}
	{attribute 'iot.MaxValue':='1200'}
	nValue			: INT;	
	nValueRequest 	: INT;
	
	sMode			: STRING; // can be set to any value, does not have to match the array below
	aModes			: ARRAY[0..1] OF STRING;
END_STRUCT
END_TYPE

// ---- DUTs/Ventilation/ST_Widget_Ventilation_Template.TcDUT
TYPE ST_Widget_Ventilation_Template :
STRUCT
	sDisplayName	: STRING := ''; // Insert STRING here to overwrite iot.DisplayName

	bOn				: BOOL;
	
	{attribute 'iot.Unit':='ppm'}
	{attribute 'iot.MinValue':='400'}
	{attribute 'iot.MaxValue':='1400'}
	nValue			: INT;	
	nValueRequest 	: INT;
	
	sMode			: STRING; // can be set to any value, does not have to match the array below
	aModes			: ARRAY[0..1] OF STRING;
END_STRUCT
END_TYPE

// ---- GVLs/GVL_Widgets.TcGVL
{attribute 'qualified_only'}
VAR_GLOBAL
		stWidgetData	: ST_WidgetData;
		stJsonData		: ST_JsonData;
END_VAR

// ---- POUs/MAIN.TcPOU
PROGRAM MAIN
VAR
	// Communicator function block with usage of SendData method
	fbIotWidgets 	: FB_IotCommunicator := 	(sHostName := '127.0.0.1',
												nPort := 1883,
												sMainTopic := 'SampleWidgets',
												sDevicename := 'Widgets Overview',
												sDeviceIcon := 'House');
	
	timer   		 : TON;
END_VAR

// Cyclic FB calling
fbIotWidgets.Execute(TRUE);

IF fbIotWidgets.bConnected THEN
	timer(IN:=TRUE, PT:=T#500MS);
END_IF

IF timer.Q THEN
	timer(IN:=FALSE);
	fbIotWidgets.SendData(ADR(GVL_Widgets.stWidgetData),SIZEOF(GVL_Widgets.stWidgetData));
END_IF

ManageWidgetsOverview();
ManageLighting();
ManageAC();
ManageBlinds();
ManageChargingStation();
ManageGeneralWidget();
ManagePlugs();
ManageRGBW();
ManageRGBWEL2564();
ManageTimeSwitch();
ManageVentilation();

WidgetValues();

METHOD ManageAC
VAR_INPUT
END_VAR
VAR
END_VAR
//Handling of commands from App
IF fbIotWidgets.fbCommand.bAvailable THEN
	//AC Sample 1 - no slider, no AC mode
	IF fbIotWidgets.fbCommand.sVarName = 'stAC.stAC1.sMode_Strength' THEN
		fbIotWidgets.fbCommand.GetValue(ADR(GVL_Widgets.stWidgetData.stAC.stAC1.sMode_Strength), SIZEOF(GVL_Widgets.stWidgetData.stAC.stAC1.sMode_Strength), E_IotCommunicatorDatatype.type_STRING);
	ELSIF fbIotWidgets.fbCommand.sVarName = 'stAC.stAC1.sMode_Lamella' THEN
		fbIotWidgets.fbCommand.GetValue(ADR(GVL_Widgets.stWidgetData.stAC.stAC1.sMode_Lamella), SIZEOF(GVL_Widgets.stWidgetData.stAC.stAC1.sMode_Lamella), E_IotCommunicatorDatatype.type_STRING);
	//AC Sample 2
	ELSIF fbIotWidgets.fbCommand.sVarName = 'stAC.stAC2.nTemperatureRequest' THEN
		fbIotWidgets.fbCommand.GetValue(ADR(GVL_Widgets.stWidgetData.stAC.stAC2.nTemperatureRequest), SIZEOF(GVL_Widgets.stWidgetData.stAC.stAC2.nTemperatureRequest), E_IotCommunicatorDatatype.type_LREAL);
	ELSIF fbIotWidgets.fbCommand.sVarName = 'stAC.stAC2.sMode' THEN
		fbIotWidgets.fbCommand.GetValue(ADR(GVL_Widgets.stWidgetData.stAC.stAC2.sMode), SIZEOF(GVL_Widgets.stWidgetData.stAC.stAC2.sMode), E_IotCommunicatorDatatype.type_STRING);
	ELSIF fbIotWidgets.fbCommand.sVarName = 'stAC.stAC2.sMode_Strength' THEN
		fbIotWidgets.fbCommand.GetValue(ADR(GVL_Widgets.stWidgetData.stAC.stAC2.sMode_Strength), SIZEOF(GVL_Widgets.stWidgetData.stAC.stAC2.sMode_Strength), E_IotCommunicatorDatatype.type_STRING);
	ELSIF fbIotWidgets.fbCommand.sVarName = 'stAC.stAC2.sMode_Lamella' THEN
		fbIotWidgets.fbCommand.GetValue(ADR(GVL_Widgets.stWidgetData.stAC.stAC2.sMode_Lamella), SIZEOF(GVL_Widgets.stWidgetData.stAC.stAC2.sMode_Lamella), E_IotCommunicatorDatatype.type_STRING);
	ELSE
		RETURN;
	END_IF
	//AC Sample 3 - no processing required - readOnly widget
	fbIotWidgets.SendData(ADR(GVL_Widgets.stWidgetData), SIZEOF(GVL_Widgets.stWidgetData));
	fbIotWidgets.fbCommand.Remove();
END_IF
END_METHOD

METHOD ManageBlinds
VAR_INPUT
END_VAR
VAR
END_VAR
//Handling of commands from App
IF fbIotWidgets.fbCommand.bAvailable THEN
	//Blinds Sample 1 - no processing required - readOnly Widget
	//Blinds Sample 2 - no mode, no angle slider/value
	IF fbIotWidgets.fbCommand.sVarName = 'stBlinds.stBlinds2.bPositionUp' THEN
		fbIotWidgets.fbCommand.GetValue(ADR(GVL_Widgets.stWidgetData.stBlinds.stBlinds2.bPositionUp), SIZEOF(GVL_Widgets.stWidgetData.stBlinds.stBlinds2.bPositionUp), E_IotCommunicatorDatatype.type_BOOL);
	ELSIF fbIotWidgets.fbCommand.sVarName = 'stBlinds.stBlinds2.bPositionDown' THEN
		fbIotWidgets.fbCommand.GetValue(ADR(GVL_Widgets.stWidgetData.stBlinds.stBlinds2.bPositionDown), SIZEOF(GVL_Widgets.stWidgetData.stBlinds.stBlinds2.bPositionDown), E_IotCommunicatorDatatype.type_BOOL);
	ELSIF fbIotWidgets.fbCommand.sVarName = 'stBlinds.stBlinds2.nPositionRequest' THEN
		fbIotWidgets.fbCommand.GetValue(ADR(GVL_Widgets.stWidgetData.stBlinds.stBlinds2.nPositionRequest), SIZEOF(GVL_Widgets.stWidgetData.stBlinds.stBlinds2.nPositionRequest), E_IotCommunicatorDatatype.type_INT);
	ELSIF fbIotWidgets.fbCommand.sVarName = 'stBlinds.stBlinds2.bActive' THEN
		fbIotWidgets.fbCommand.GetValue(ADR(GVL_Widgets.stWidgetData.stBlinds.stBlinds2.bActive), SIZEOF(GVL_Widgets.stWidgetData.stBlinds.stBlinds2.bActive), E_IotCommunicatorDatatype.type_BOOL);
	//Blinds Sample 3
	ELSIF fbIotWidgets.fbCommand.sVarName = 'stBlinds.stBlinds3.bPositionUp' THEN
		fbIotWidgets.fbCommand.GetValue(ADR(GVL_Widgets.stWidgetData.stBlinds.stBlinds3.bPositionUp), SIZEOF(GVL_Widgets.stWidgetData.stBlinds.stBlinds3.bPositionUp), E_IotCommunicatorDatatype.type_BOOL);
	ELSIF fbIotWidgets.fbCommand.sVarName = 'stBlinds.stBlinds3.bPositionDown' THEN
		fbIotWidgets.fbCommand.GetValue(ADR(GVL_Widgets.stWidgetData.stBlinds.stBlinds3.bPositionDown), SIZEOF(GVL_Widgets.stWidgetData.stBlinds.stBlinds3.bPositionDown), E_IotCommunicatorDatatype.type_BOOL);
	ELSIF fbIotWidgets.fbCommand.sVarName = 'stBlinds.stBlinds3.nPositionRequest' THEN
		fbIotWidgets.fbCommand.GetValue(ADR(GVL_Widgets.stWidgetData.stBlinds.stBlinds3.nPositionRequest), SIZEOF(GVL_Widgets.stWidgetData.stBlinds.stBlinds3.nPositionRequest), E_IotCommunicatorDatatype.type_INT);
	ELSIF fbIotWidgets.fbCommand.sVarName = 'stBlinds.stBlinds3.bAngleUp' THEN
		fbIotWidgets.fbCommand.GetValue(ADR(GVL_Widgets.stWidgetData.stBlinds.stBlinds3.bAngleUp), SIZEOF(GVL_Widgets.stWidgetData.stBlinds.stBlinds3.bAngleUp), E_IotCommunicatorDatatype.type_BOOL);
	ELSIF fbIotWidgets.fbCommand.sVarName = 'stBlinds.stBlinds3.bAngleDown' THEN
		fbIotWidgets.fbCommand.GetValue(ADR(GVL_Widgets.stWidgetData.stBlinds.stBlinds3.bAngleDown), SIZEOF(GVL_Widgets.stWidgetData.stBlinds.stBlinds3.bAngleDown), E_IotCommunicatorDatatype.type_BOOL);
	ELSIF fbIotWidgets.fbCommand.sVarName = 'stBlinds.stBlinds3.nAngleRequest' THEN
		fbIotWidgets.fbCommand.GetValue(ADR(GVL_Widgets.stWidgetData.stBlinds.stBlinds3.nAngleRequest), SIZEOF(GVL_Widgets.stWidgetData.stBlinds.stBlinds3.nAngleRequest), E_IotCommunicatorDatatype.type_INT);
	ELSIF fbIotWidgets.fbCommand.sVarName = 'stBlinds.stBlinds3.sMode' THEN
		fbIotWidgets.fbCommand.GetValue(ADR(GVL_Widgets.stWidgetData.stBlinds.stBlinds3.sMode), SIZEOF(GVL_Widgets.stWidgetData.stBlinds.stBlinds3.sMode), E_IotCommunicatorDatatype.type_STRING);
	ELSIF fbIotWidgets.fbCommand.sVarName = 'stBlinds.stBlinds3.bActive' THEN
		fbIotWidgets.fbCommand.GetValue(ADR(GVL_Widgets.stWidgetData.stBlinds.stBlinds3.bActive), SIZEOF(GVL_Widgets.stWidgetData.stBlinds.stBlinds3.bActive), E_IotCommunicatorDatatype.type_BOOL);
	//Simple Blinds Sample 1
	ELSIF fbIotWidgets.fbCommand.sVarName = 'stBlinds.stSimpleBlinds1.bPositionUp' THEN
		fbIotWidgets.fbCommand.GetValue(ADR(GVL_Widgets.stWidgetData.stBlinds.stSimpleBlinds1.bPositionUp), SIZEOF(GVL_Widgets.stWidgetData.stBlinds.stSimpleBlinds1.bPositionUp), E_IotCommunicatorDatatype.type_BOOL);
	ELSIF fbIotWidgets.fbCommand.sVarName = 'stBlinds.stSimpleBlinds1.bPositionDown' THEN
		fbIotWidgets.fbCommand.GetValue(ADR(GVL_Widgets.stWidgetData.stBlinds.stSimpleBlinds1.bPositionDown), SIZEOF(GVL_Widgets.stWidgetData.stBlinds.stSimpleBlinds1.bPositionDown), E_IotCommunicatorDatatype.type_BOOL);
	//Simple Blinds Sample 2
	ELSIF fbIotWidgets.fbCommand.sVarName = 'stBlinds.stSimpleBlinds2.bPositionUp' THEN
		fbIotWidgets.fbCommand.GetValue(ADR(GVL_Widgets.stWidgetData.stBlinds.stSimpleBlinds2.bPositionUp), SIZEOF(GVL_Widgets.stWidgetData.stBlinds.stSimpleBlinds2.bPositionUp), E_IotCommunicatorDatatype.type_BOOL);
	ELSIF fbIotWidgets.fbCommand.sVarName = 'stBlinds.stSimpleBlinds2.bPositionDown' THEN
		fbIotWidgets.fbCommand.GetValue(ADR(GVL_Widgets.stWidgetData.stBlinds.stSimpleBlinds2.bPositionDown), SIZEOF(GVL_Widgets.stWidgetData.stBlinds.stSimpleBlinds2.bPositionDown), E_IotCommunicatorDatatype.type_BOOL);
	ELSE
		RETURN;
	END_IF
	fbIotWidgets.SendData(ADR(GVL_Widgets.stWidgetData), SIZEOF(GVL_Widgets.stWidgetData));
	fbIotWidgets.fbCommand.Remove();
END_IF
END_METHOD

METHOD ManageChargingStation
VAR_INPUT
END_VAR
//Handling of commands from App
IF fbIotWidgets.fbCommand.bAvailable THEN
	// Charging Station Sample 1 - Receive Start, Stop, Reserve requests
	IF fbIotWidgets.fbCommand.sVarName = 'stChargingStation.stChargingStation1.bStartCharging' THEN
		fbIotWidgets.fbCommand.GetValue(ADR(GVL_Widgets.stWidgetData.stChargingStation.stChargingStation1.bStartCharging), SIZEOF(GVL_Widgets.stWidgetData.stChargingStation.stChargingStation1.bStartCharging), E_IotCommunicatorDatatype.type_BOOL);
	ELSIF fbIotWidgets.fbCommand.sVarName = 'stChargingStation.stChargingStation1.bStopCharging' THEN
		fbIotWidgets.fbCommand.GetValue(ADR(GVL_Widgets.stWidgetData.stChargingStation.stChargingStation1.bStopCharging), SIZEOF(GVL_Widgets.stWidgetData.stChargingStation.stChargingStation1.bStopCharging), E_IotCommunicatorDatatype.type_BOOL);
	ELSIF fbIotWidgets.fbCommand.sVarName = 'stChargingStation.stChargingStation1.bReserveCharging' THEN
		fbIotWidgets.fbCommand.GetValue(ADR(GVL_Widgets.stWidgetData.stChargingStation.stChargingStation1.bReserveCharging), SIZEOF(GVL_Widgets.stWidgetData.stChargingStation.stChargingStation1.bReserveCharging), E_IotCommunicatorDatatype.type_BOOL);
	ELSIF fbIotWidgets.fbCommand.sVarName = 'stChargingStation.stChargingStation2.bStartCharging' THEN
		fbIotWidgets.fbCommand.GetValue(ADR(GVL_Widgets.stWidgetData.stChargingStation.stChargingStation2.bStartCharging), SIZEOF(GVL_Widgets.stWidgetData.stChargingStation.stChargingStation2.bStartCharging), E_IotCommunicatorDatatype.type_BOOL);
	ELSIF fbIotWidgets.fbCommand.sVarName = 'stChargingStation.stChargingStation2.bStopCharging' THEN
		fbIotWidgets.fbCommand.GetValue(ADR(GVL_Widgets.stWidgetData.stChargingStation.stChargingStation2.bStopCharging), SIZEOF(GVL_Widgets.stWidgetData.stChargingStation.stChargingStation2.bStopCharging), E_IotCommunicatorDatatype.type_BOOL);
	ELSE
		RETURN;
	END_IF	
	fbIotWidgets.SendData(ADR(GVL_Widgets.stWidgetData), SIZEOF(GVL_Widgets.stWidgetData));
	fbIotWidgets.fbCommand.Remove();
END_IF
END_METHOD

METHOD ManageGeneralWidget
VAR_INPUT
END_VAR
VAR
END_VAR
//Handling of commands from App
IF fbIotWidgets.fbCommand.bAvailable THEN
	//General Widget Sample 1 - no processing required - readOnly Widget
	//General Widget Sample 2 - two modes, one slider
	IF fbIotWidgets.fbCommand.sVarName = 'stGeneral.stGeneral2.bValue1' THEN
		fbIotWidgets.fbCommand.GetValue(ADR(GVL_Widgets.stWidgetData.stGeneral.stGeneral2.bValue1), SIZEOF(GVL_Widgets.stWidgetData.stGeneral.stGeneral2.bValue1), E_IotCommunicatorDatatype.type_BOOL);
	ELSIF fbIotWidgets.fbCommand.sVarName = 'stGeneral.stGeneral2.bValue2Up' THEN
		fbIotWidgets.fbCommand.GetValue(ADR(GVL_Widgets.stWidgetData.stGeneral.stGeneral2.bValue2Up), SIZEOF(GVL_Widgets.stWidgetData.stGeneral.stGeneral2.bValue2Up), E_IotCommunicatorDatatype.type_BOOL);
	ELSIF fbIotWidgets.fbCommand.sVarName = 'stGeneral.stGeneral2.bValue2Down' THEN
		fbIotWidgets.fbCommand.GetValue(ADR(GVL_Widgets.stWidgetData.stGeneral.stGeneral2.bValue2Down), SIZEOF(GVL_Widgets.stWidgetData.stGeneral.stGeneral2.bValue2Down), E_IotCommunicatorDatatype.type_BOOL);
	ELSIF fbIotWidgets.fbCommand.sVarName = 'stGeneral.stGeneral2.nValue2Request' THEN
		fbIotWidgets.fbCommand.GetValue(ADR(GVL_Widgets.stWidgetData.stGeneral.stGeneral2.nValue2Request), SIZEOF(GVL_Widgets.stWidgetData.stGeneral.stGeneral2.nValue2Request), E_IotCommunicatorDatatype.type_INT);
	ELSIF fbIotWidgets.fbCommand.sVarName = 'stGeneral.stGeneral2.sMode1' THEN
		fbIotWidgets.fbCommand.GetValue(ADR(GVL_Widgets.stWidgetData.stGeneral.stGeneral2.sMode1), SIZEOF(GVL_Widgets.stWidgetData.stGeneral.stGeneral2.sMode1), E_IotCommunicatorDatatype.type_STRING);
	//General Widget Sample 3
	ELSIF fbIotWidgets.fbCommand.sVarName = 'stGeneral.stGeneral3.bValue1' THEN
		fbIotWidgets.fbCommand.GetValue(ADR(GVL_Widgets.stWidgetData.stGeneral.stGeneral3.bValue1), SIZEOF(GVL_Widgets.stWidgetData.stGeneral.stGeneral3.bValue1), E_IotCommunicatorDatatype.type_BOOL);
	ELSIF fbIotWidgets.fbCommand.sVarName = 'stGeneral.stGeneral3.bValue2Up' THEN
		fbIotWidgets.fbCommand.GetValue(ADR(GVL_Widgets.stWidgetData.stGeneral.stGeneral3.bValue2Up), SIZEOF(GVL_Widgets.stWidgetData.stGeneral.stGeneral3.bValue2Up), E_IotCommunicatorDatatype.type_BOOL);
	ELSIF fbIotWidgets.fbCommand.sVarName = 'stGeneral.stGeneral3.bValue2Down' THEN
		fbIotWidgets.fbCommand.GetValue(ADR(GVL_Widgets.stWidgetData.stGeneral.stGeneral3.bValue2Down), SIZEOF(GVL_Widgets.stWidgetData.stGeneral.stGeneral3.bValue2Down), E_IotCommunicatorDatatype.type_BOOL);
	ELSIF fbIotWidgets.fbCommand.sVarName = 'stGeneral.stGeneral3.nValue2Request' THEN
		fbIotWidgets.fbCommand.GetValue(ADR(GVL_Widgets.stWidgetData.stGeneral.stGeneral3.nValue2Request), SIZEOF(GVL_Widgets.stWidgetData.stGeneral.stGeneral3.nValue2Request), E_IotCommunicatorDatatype.type_INT);
	ELSIF fbIotWidgets.fbCommand.sVarName = 'stGeneral.stGeneral3.bValue3Up' THEN
		fbIotWidgets.fbCommand.GetValue(ADR(GVL_Widgets.stWidgetData.stGeneral.stGeneral3.bValue3Up), SIZEOF(GVL_Widgets.stWidgetData.stGeneral.stGeneral3.bValue3Up), E_IotCommunicatorDatatype.type_BOOL);
	ELSIF fbIotWidgets.fbCommand.sVarName = 'stGeneral.stGeneral3.bValue3Down' THEN
		fbIotWidgets.fbCommand.GetValue(ADR(GVL_Widgets.stWidgetData.stGeneral.stGeneral3.bValue3Down), SIZEOF(GVL_Widgets.stWidgetData.stGeneral.stGeneral3.bValue3Down), E_IotCommunicatorDatatype.type_BOOL);
	ELSIF fbIotWidgets.fbCommand.sVarName = 'stGeneral.stGeneral3.nValue3Request' THEN
		fbIotWidgets.fbCommand.GetValue(ADR(GVL_Widgets.stWidgetData.stGeneral.stGeneral3.nValue3Request), SIZEOF(GVL_Widgets.stWidgetData.stGeneral.stGeneral3.nValue3Request), E_IotCommunicatorDatatype.type_INT);
	ELSIF fbIotWidgets.fbCommand.sVarName = 'stGeneral.stGeneral3.sMode1' THEN
		fbIotWidgets.fbCommand.GetValue(ADR(GVL_Widgets.stWidgetData.stGeneral.stGeneral3.sMode1), SIZEOF(GVL_Widgets.stWidgetData.stGeneral.stGeneral3.sMode1), E_IotCommunicatorDatatype.type_STRING);
	ELSIF fbIotWidgets.fbCommand.sVarName = 'stGeneral.stGeneral3.sMode2' THEN
		fbIotWidgets.fbCommand.GetValue(ADR(GVL_Widgets.stWidgetData.stGeneral.stGeneral3.sMode2), SIZEOF(GVL_Widgets.stWidgetData.stGeneral.stGeneral3.sMode2), E_IotCommunicatorDatatype.type_STRING);
	ELSIF fbIotWidgets.fbCommand.sVarName = 'stGeneral.stGeneral3.sMode3' THEN
		fbIotWidgets.fbCommand.GetValue(ADR(GVL_Widgets.stWidgetData.stGeneral.stGeneral3.sMode3), SIZEOF(GVL_Widgets.stWidgetData.stGeneral.stGeneral3.sMode3), E_IotCommunicatorDatatype.type_STRING);
	ELSE
		RETURN;
	END_IF
	fbIotWidgets.SendData(ADR(GVL_Widgets.stWidgetData), SIZEOF(GVL_Widgets.stWidgetData));
	fbIotWidgets.fbCommand.Remove();
END_IF
END_METHOD

METHOD ManageLighting
VAR_INPUT
END_VAR
VAR
END_VAR
//Handling of commands from App
IF fbIotWidgets.fbCommand.bAvailable THEN
	//Lighting Sample 1 - no processing required - readOnly Widget
	//Lighting Sample 2 - no value
	IF fbIotWidgets.fbCommand.sVarName = 'stLights.stLighting2.bLight' THEN
		fbIotWidgets.fbCommand.GetValue(ADR(GVL_Widgets.stWidgetData.stLights.stLighting2.bLight), SIZEOF(GVL_Widgets.stWidgetData.stLights.stLighting2.bLight), E_IotCommunicatorDatatype.type_BOOL);
	ELSIF fbIotWidgets.fbCommand.sVarName = 'stLights.stLighting2.nLight' THEN
		fbIotWidgets.fbCommand.GetValue(ADR(GVL_Widgets.stWidgetData.stLights.stLighting2.nLight), SIZEOF(GVL_Widgets.stWidgetData.stLights.stLighting2.nLight), E_IotCommunicatorDatatype.type_INT);
	ELSIF fbIotWidgets.fbCommand.sVarName = 'stLights.stLighting2.sMode' THEN
		fbIotWidgets.fbCommand.GetValue(ADR(GVL_Widgets.stWidgetData.stLights.stLighting2.sMode), SIZEOF(GVL_Widgets.stWidgetData.stLights.stLighting2.sMode), E_IotCommunicatorDatatype.type_STRING);
	//Lighting Sample 3
	ELSIF fbIotWidgets.fbCommand.sVarName = 'stLights.stLighting3.bLight' THEN
		fbIotWidgets.fbCommand.GetValue(ADR(GVL_Widgets.stWidgetData.stLights.stLighting3.bLight), SIZEOF(GVL_Widgets.stWidgetData.stLights.stLighting3.bLight), E_IotCommunicatorDatatype.type_BOOL);
	ELSIF fbIotWidgets.fbCommand.sVarName = 'stLights.stLighting3.nLight' THEN
		fbIotWidgets.fbCommand.GetValue(ADR(GVL_Widgets.stWidgetData.stLights.stLighting3.nLight), SIZEOF(GVL_Widgets.stWidgetData.stLights.stLighting3.nLight), E_IotCommunicatorDatatype.type_INT);
	ELSIF fbIotWidgets.fbCommand.sVarName = 'stLights.stLighting3.sMode' THEN
		fbIotWidgets.fbCommand.GetValue(ADR(GVL_Widgets.stWidgetData.stLights.stLighting3.sMode), SIZEOF(GVL_Widgets.stWidgetData.stLights.stLighting3.sMode), E_IotCommunicatorDatatype.type_STRING);
	ELSE
		RETURN;
	END_IF
	fbIotWidgets.SendData(ADR(GVL_Widgets.stWidgetData), SIZEOF(GVL_Widgets.stWidgetData));
	fbIotWidgets.fbCommand.Remove();
END_IF

//Lighting Sample 2
GVL_Widgets.stWidgetData.stLights.stLighting2.aModes[0]:='Automatic';
GVL_Widgets.stWidgetData.stLights.stLighting2.aModes[1]:='Manual';
//Lighting Sample 3
GVL_Widgets.stWidgetData.stLights.stLighting3.aModes[0]:='Night';
GVL_Widgets.stWidgetData.stLights.stLighting3.aModes[1]:='Day';
END_METHOD

METHOD ManagePlugs
VAR_INPUT
END_VAR
VAR
END_VAR
//Handling of commands from App
IF fbIotWidgets.fbCommand.bAvailable THEN
	//Plug Sample 1 - no mode
	IF fbIotWidgets.fbCommand.sVarName = 'stPlugs.stPlug1.bOn' THEN
		fbIotWidgets.fbCommand.GetValue(ADR(GVL_Widgets.stWidgetData.stPlugs.stPlug1.bOn), SIZEOF(GVL_Widgets.stWidgetData.stPlugs.stPlug1.bOn), E_IotCommunicatorDatatype.type_BOOL);
	//Plug Sample 2
	ELSIF fbIotWidgets.fbCommand.sVarName = 'stPlugs.stPlug2.bOn' THEN
		fbIotWidgets.fbCommand.GetValue(ADR(GVL_Widgets.stWidgetData.stPlugs.stPlug2.bOn), SIZEOF(GVL_Widgets.stWidgetData.stPlugs.stPlug2.bOn), E_IotCommunicatorDatatype.type_BOOL);
	ELSIF fbIotWidgets.fbCommand.sVarName = 'stPlugs.stPlug2.sMode' THEN
		fbIotWidgets.fbCommand.GetValue(ADR(GVL_Widgets.stWidgetData.stPlugs.stPlug2.sMode), SIZEOF(GVL_Widgets.stWidgetData.stPlugs.stPlug2.sMode), E_IotCommunicatorDatatype.type_STRING);
	ELSE
		RETURN;
	END_IF
	fbIotWidgets.SendData(ADR(GVL_Widgets.stWidgetData), SIZEOF(GVL_Widgets.stWidgetData));
	fbIotWidgets.fbCommand.Remove();
END_IF
END_METHOD

METHOD ManageRGBW
VAR_INPUT
END_VAR
//Handling of commands from App
IF fbIotWidgets.fbCommand.bAvailable THEN
	//RGBW Sample 2 - no color temperature
	IF fbIotWidgets.fbCommand.sVarName = 'stRGBW.stRGB2.bLight' THEN
		fbIotWidgets.fbCommand.GetValue(ADR(GVL_Widgets.stWidgetData.stRGBW.stRGB2.bLight), SIZEOF(GVL_Widgets.stWidgetData.stRGBW.stRGB2.bLight), E_IotCommunicatorDatatype.type_BOOL);
	ELSIF fbIotWidgets.fbCommand.sVarName = 'stRGBW.stRGB2.nLight' THEN
		fbIotWidgets.fbCommand.GetValue(ADR(GVL_Widgets.stWidgetData.stRGBW.stRGB2.nLight), SIZEOF(GVL_Widgets.stWidgetData.stRGBW.stRGB2.nLight), E_IotCommunicatorDatatype.type_INT);
	ELSIF fbIotWidgets.fbCommand.sVarName = 'stRGBW.stRGB2.nHueValue' THEN
		fbIotWidgets.fbCommand.GetValue(ADR(GVL_Widgets.stWidgetData.stRGBW.stRGB2.nHueValue), SIZEOF(GVL_Widgets.stWidgetData.stRGBW.stRGB2.nHueValue), E_IotCommunicatorDatatype.type_INT);
	ELSIF fbIotWidgets.fbCommand.sVarName = 'stRGBW.stRGB2.nSaturation' THEN
		fbIotWidgets.fbCommand.GetValue(ADR(GVL_Widgets.stWidgetData.stRGBW.stRGB2.nSaturation), SIZEOF(GVL_Widgets.stWidgetData.stRGBW.stRGB2.nSaturation), E_IotCommunicatorDatatype.type_INT);
	ELSIF fbIotWidgets.fbCommand.sVarName = 'stRGBW.stRGB2.sMode' THEN
		fbIotWidgets.fbCommand.GetValue(ADR(GVL_Widgets.stWidgetData.stRGBW.stRGB2.sMode), SIZEOF(GVL_Widgets.stWidgetData.stRGBW.stRGB2.sMode), E_IotCommunicatorDatatype.type_STRING);
	//RGBW Sample 3
	ELSIF fbIotWidgets.fbCommand.sVarName = 'stRGBW.stRGB3.bLight' THEN
		fbIotWidgets.fbCommand.GetValue(ADR(GVL_Widgets.stWidgetData.stRGBW.stRGB3.bLight), SIZEOF(GVL_Widgets.stWidgetData.stRGBW.stRGB3.bLight), E_IotCommunicatorDatatype.type_BOOL);
	ELSIF fbIotWidgets.fbCommand.sVarName = 'stRGBW.stRGB3.nLight' THEN
		fbIotWidgets.fbCommand.GetValue(ADR(GVL_Widgets.stWidgetData.stRGBW.stRGB3.nLight), SIZEOF(GVL_Widgets.stWidgetData.stRGBW.stRGB3.nLight), E_IotCommunicatorDatatype.type_INT);
	ELSIF fbIotWidgets.fbCommand.sVarName = 'stRGBW.stRGB3.nHueValue' THEN
		fbIotWidgets.fbCommand.GetValue(ADR(GVL_Widgets.stWidgetData.stRGBW.stRGB3.nHueValue), SIZEOF(GVL_Widgets.stWidgetData.stRGBW.stRGB3.nHueValue), E_IotCommunicatorDatatype.type_INT);
	ELSIF fbIotWidgets.fbCommand.sVarName = 'stRGBW.stRGB3.nSaturation' THEN
		fbIotWidgets.fbCommand.GetValue(ADR(GVL_Widgets.stWidgetData.stRGBW.stRGB3.nSaturation), SIZEOF(GVL_Widgets.stWidgetData.stRGBW.stRGB3.nSaturation), E_IotCommunicatorDatatype.type_INT);
	ELSIF fbIotWidgets.fbCommand.sVarName = 'stRGBW.stRGB3.nColorTemperature' THEN
		fbIotWidgets.fbCommand.GetValue(ADR(GVL_Widgets.stWidgetData.stRGBW.stRGB3.nColorTemperature), SIZEOF(GVL_Widgets.stWidgetData.stRGBW.stRGB3.nColorTemperature), E_IotCommunicatorDatatype.type_INT);
	ELSIF fbIotWidgets.fbCommand.sVarName = 'stRGBW.stRGB3.nWhite' THEN
		fbIotWidgets.fbCommand.GetValue(ADR(GVL_Widgets.stWidgetData.stRGBW.stRGB3.nWhite), SIZEOF(GVL_Widgets.stWidgetData.stRGBW.stRGB3.nWhite), E_IotCommunicatorDatatype.type_INT);
	ELSIF fbIotWidgets.fbCommand.sVarName = 'stRGBW.stRGB3.sMode' THEN
		fbIotWidgets.fbCommand.GetValue(ADR(GVL_Widgets.stWidgetData.stRGBW.stRGB3.sMode), SIZEOF(GVL_Widgets.stWidgetData.stRGBW.stRGB3.sMode), E_IotCommunicatorDatatype.type_STRING);
	ELSE
		RETURN;
	END_IF
	fbIotWidgets.SendData(ADR(GVL_Widgets.stWidgetData), SIZEOF(GVL_Widgets.stWidgetData));
	fbIotWidgets.fbCommand.Remove();
END_IF
END_METHOD

METHOD ManageRGBWEL2564
VAR_INPUT
END_VAR
//Handling of commands from App
IF fbIotWidgets.fbCommand.bAvailable THEN
	//RGBW EL2564 Sample 2 - no modes
	IF fbIotWidgets.fbCommand.sVarName = 'stRGBWEL2564.stRGBWLed2.bOn' THEN
		fbIotWidgets.fbCommand.GetValue(ADR(GVL_Widgets.stWidgetData.stRGBWEL2564.stRGBWLed2.bOn), SIZEOF(GVL_Widgets.stWidgetData.stRGBWEL2564.stRGBWLed2.bOn), E_IotCommunicatorDatatype.type_BOOL);
	ELSIF fbIotWidgets.fbCommand.sVarName = 'stRGBWEL2564.stRGBWLed2.nGreen' THEN
		fbIotWidgets.fbCommand.GetValue(ADR(GVL_Widgets.stWidgetData.stRGBWEL2564.stRGBWLed2.nGreen), SIZEOF(GVL_Widgets.stWidgetData.stRGBWEL2564.stRGBWLed2.nGreen), E_IotCommunicatorDatatype.type_INT);
	ELSIF fbIotWidgets.fbCommand.sVarName = 'stRGBWEL2564.stRGBWLed2.nBlue' THEN
		fbIotWidgets.fbCommand.GetValue(ADR(GVL_Widgets.stWidgetData.stRGBWEL2564.stRGBWLed2.nBlue), SIZEOF(GVL_Widgets.stWidgetData.stRGBWEL2564.stRGBWLed2.nBlue), E_IotCommunicatorDatatype.type_INT);
	ELSIF fbIotWidgets.fbCommand.sVarName = 'stRGBWEL2564.stRGBWLed2.nRed' THEN
		fbIotWidgets.fbCommand.GetValue(ADR(GVL_Widgets.stWidgetData.stRGBWEL2564.stRGBWLed2.nRed), SIZEOF(GVL_Widgets.stWidgetData.stRGBWEL2564.stRGBWLed2.nRed), E_IotCommunicatorDatatype.type_INT);
	ELSIF fbIotWidgets.fbCommand.sVarName = 'stRGBWEL2564.stRGBWLed2.nWhite' THEN
		fbIotWidgets.fbCommand.GetValue(ADR(GVL_Widgets.stWidgetData.stRGBWEL2564.stRGBWLed2.nWhite), SIZEOF(GVL_Widgets.stWidgetData.stRGBWEL2564.stRGBWLed2.nWhite), E_IotCommunicatorDatatype.type_INT);
	ELSIF fbIotWidgets.fbCommand.sVarName = 'stRGBWEL2564.stRGBWLed2.sMode' THEN
		fbIotWidgets.fbCommand.GetValue(ADR(GVL_Widgets.stWidgetData.stRGBWEL2564.stRGBWLed2.sMode), SIZEOF(GVL_Widgets.stWidgetData.stRGBWEL2564.stRGBWLed2.sMode), E_IotCommunicatorDatatype.type_STRING);
	//RGBW EL2564 Sample 3
	ELSIF fbIotWidgets.fbCommand.sVarName = 'stRGBWEL2564.stRGBWLed3.bOn' THEN
		fbIotWidgets.fbCommand.GetValue(ADR(GVL_Widgets.stWidgetData.stRGBWEL2564.stRGBWLed3.bOn), SIZEOF(GVL_Widgets.stWidgetData.stRGBWEL2564.stRGBWLed3.bOn), E_IotCommunicatorDatatype.type_BOOL);
	ELSIF fbIotWidgets.fbCommand.sVarName = 'stRGBWEL2564.stRGBWLed3.nGreen' THEN
		fbIotWidgets.fbCommand.GetValue(ADR(GVL_Widgets.stWidgetData.stRGBWEL2564.stRGBWLed3.nGreen), SIZEOF(GVL_Widgets.stWidgetData.stRGBWEL2564.stRGBWLed3.nGreen), E_IotCommunicatorDatatype.type_INT);
	ELSIF fbIotWidgets.fbCommand.sVarName = 'stRGBWEL2564.stRGBWLed3.nBlue' THEN
		fbIotWidgets.fbCommand.GetValue(ADR(GVL_Widgets.stWidgetData.stRGBWEL2564.stRGBWLed3.nBlue), SIZEOF(GVL_Widgets.stWidgetData.stRGBWEL2564.stRGBWLed3.nBlue), E_IotCommunicatorDatatype.type_INT);
	ELSIF fbIotWidgets.fbCommand.sVarName = 'stRGBWEL2564.stRGBWLed3.nRed' THEN
		fbIotWidgets.fbCommand.GetValue(ADR(GVL_Widgets.stWidgetData.stRGBWEL2564.stRGBWLed3.nRed), SIZEOF(GVL_Widgets.stWidgetData.stRGBWEL2564.stRGBWLed3.nRed), E_IotCommunicatorDatatype.type_INT);
	ELSIF fbIotWidgets.fbCommand.sVarName = 'stRGBWEL2564.stRGBWLed3.nWhite' THEN
		fbIotWidgets.fbCommand.GetValue(ADR(GVL_Widgets.stWidgetData.stRGBWEL2564.stRGBWLed3.nWhite), SIZEOF(GVL_Widgets.stWidgetData.stRGBWEL2564.stRGBWLed3.nWhite), E_IotCommunicatorDatatype.type_INT);
	ELSIF fbIotWidgets.fbCommand.sVarName = 'stRGBWEL2564.stRGBWLed3.sMode' THEN
		fbIotWidgets.fbCommand.GetValue(ADR(GVL_Widgets.stWidgetData.stRGBWEL2564.stRGBWLed3.sMode), SIZEOF(GVL_Widgets.stWidgetData.stRGBWEL2564.stRGBWLed3.sMode), E_IotCommunicatorDatatype.type_STRING);
	ELSE
		RETURN;
	END_IF
	fbIotWidgets.SendData(ADR(GVL_Widgets.stWidgetData), SIZEOF(GVL_Widgets.stWidgetData));
	fbIotWidgets.fbCommand.Remove();
END_IF
END_METHOD

METHOD ManageTimeSwitch
VAR_INPUT
END_VAR
VAR
END_VAR
//Handling of commands from App
IF fbIotWidgets.fbCommand.bAvailable THEN
	//TimeSwitch Sample 1 - no days visible, mode readOnly
	IF fbIotWidgets.fbCommand.sVarName = 'stTimeSwitch.stTimeSwitch1.bOn' THEN
		fbIotWidgets.fbCommand.GetValue(ADR(GVL_Widgets.stWidgetData.stTimeSwitch.stTimeSwitch1.bOn), SIZEOF(GVL_Widgets.stWidgetData.stTimeSwitch.stTimeSwitch1.bOn), E_IotCommunicatorDatatype.type_BOOL);
	ELSIF fbIotWidgets.fbCommand.sVarName = 'stTimeSwitch.stTimeSwitch1.bYearly' THEN
		fbIotWidgets.fbCommand.GetValue(ADR(GVL_Widgets.stWidgetData.stTimeSwitch.stTimeSwitch1.bYearly), SIZEOF(GVL_Widgets.stWidgetData.stTimeSwitch.stTimeSwitch1.bYearly), E_IotCommunicatorDatatype.type_BOOL);
	ELSIF fbIotWidgets.fbCommand.sVarName = 'stTimeSwitch.stTimeSwitch1.tStartTime' THEN
		fbIotWidgets.fbCommand.GetValue(ADR(GVL_Widgets.stWidgetData.stTimeSwitch.stTimeSwitch1.tStartTime), SIZEOF(GVL_Widgets.stWidgetData.stTimeSwitch.stTimeSwitch1.tStartTime), E_IotCommunicatorDatatype.type_TIME_OF_DAY);
	ELSIF fbIotWidgets.fbCommand.sVarName = 'stTimeSwitch.stTimeSwitch1.tEndTime' THEN
		fbIotWidgets.fbCommand.GetValue(ADR(GVL_Widgets.stWidgetData.stTimeSwitch.stTimeSwitch1.tEndTime), SIZEOF(GVL_Widgets.stWidgetData.stTimeSwitch.stTimeSwitch1.tEndTime), E_IotCommunicatorDatatype.type_TIME_OF_DAY);
	ELSIF fbIotWidgets.fbCommand.sVarName = 'stTimeSwitch.stTimeSwitch1.dStartDate' THEN
		fbIotWidgets.fbCommand.GetValue(ADR(GVL_Widgets.stWidgetData.stTimeSwitch.stTimeSwitch1.dStartDate), SIZEOF(GVL_Widgets.stWidgetData.stTimeSwitch.stTimeSwitch1.dStartDate), E_IotCommunicatorDatatype.type_DATE);
	ELSIF fbIotWidgets.fbCommand.sVarName = 'stTimeSwitch.stTimeSwitch1.dEndDate' THEN
		fbIotWidgets.fbCommand.GetValue(ADR(GVL_Widgets.stWidgetData.stTimeSwitch.stTimeSwitch1.dEndDate), SIZEOF(GVL_Widgets.stWidgetData.stTimeSwitch.stTimeSwitch1.dEndDate), E_IotCommunicatorDatatype.type_DATE);
	//TimeSwitch Sample 2 - no dates visible, no mode
	ELSIF fbIotWidgets.fbCommand.sVarName = 'stTimeSwitch.stTimeSwitch2.bOn' THEN
		fbIotWidgets.fbCommand.GetValue(ADR(GVL_Widgets.stWidgetData.stTimeSwitch.stTimeSwitch2.bOn), SIZEOF(GVL_Widgets.stWidgetData.stTimeSwitch.stTimeSwitch2.bOn), E_IotCommunicatorDatatype.type_BOOL);
	ELSIF fbIotWidgets.fbCommand.sVarName = 'stTimeSwitch.stTimeSwitch2.bYearly' THEN
		fbIotWidgets.fbCommand.GetValue(ADR(GVL_Widgets.stWidgetData.stTimeSwitch.stTimeSwitch2.bYearly), SIZEOF(GVL_Widgets.stWidgetData.stTimeSwitch.stTimeSwitch2.bYearly), E_IotCommunicatorDatatype.type_BOOL);
	ELSIF fbIotWidgets.fbCommand.sVarName = 'stTimeSwitch.stTimeSwitch2.bMonday' THEN
		fbIotWidgets.fbCommand.GetValue(ADR(GVL_Widgets.stWidgetData.stTimeSwitch.stTimeSwitch2.bMonday), SIZEOF(GVL_Widgets.stWidgetData.stTimeSwitch.stTimeSwitch2.bMonday), E_IotCommunicatorDatatype.type_BOOL);
	ELSIF fbIotWidgets.fbCommand.sVarName = 'stTimeSwitch.stTimeSwitch2.bTuesday' THEN
		fbIotWidgets.fbCommand.GetValue(ADR(GVL_Widgets.stWidgetData.stTimeSwitch.stTimeSwitch2.bTuesday), SIZEOF(GVL_Widgets.stWidgetData.stTimeSwitch.stTimeSwitch2.bTuesday), E_IotCommunicatorDatatype.type_BOOL);
	ELSIF fbIotWidgets.fbCommand.sVarName = 'stTimeSwitch.stTimeSwitch2.bWednesday' THEN
		fbIotWidgets.fbCommand.GetValue(ADR(GVL_Widgets.stWidgetData.stTimeSwitch.stTimeSwitch2.bWednesday), SIZEOF(GVL_Widgets.stWidgetData.stTimeSwitch.stTimeSwitch2.bWednesday), E_IotCommunicatorDatatype.type_BOOL);
	ELSIF fbIotWidgets.fbCommand.sVarName = 'stTimeSwitch.stTimeSwitch2.bThursday' THEN
		fbIotWidgets.fbCommand.GetValue(ADR(GVL_Widgets.stWidgetData.stTimeSwitch.stTimeSwitch2.bThursday), SIZEOF(GVL_Widgets.stWidgetData.stTimeSwitch.stTimeSwitch2.bThursday), E_IotCommunicatorDatatype.type_BOOL);
	ELSIF fbIotWidgets.fbCommand.sVarName = 'stTimeSwitch.stTimeSwitch2.bFriday' THEN
		fbIotWidgets.fbCommand.GetValue(ADR(GVL_Widgets.stWidgetData.stTimeSwitch.stTimeSwitch2.bFriday), SIZEOF(GVL_Widgets.stWidgetData.stTimeSwitch.stTimeSwitch2.bFriday), E_IotCommunicatorDatatype.type_BOOL);
	ELSIF fbIotWidgets.fbCommand.sVarName = 'stTimeSwitch.stTimeSwitch2.bSaturday' THEN
		fbIotWidgets.fbCommand.GetValue(ADR(GVL_Widgets.stWidgetData.stTimeSwitch.stTimeSwitch2.bSaturday), SIZEOF(GVL_Widgets.stWidgetData.stTimeSwitch.stTimeSwitch2.bSaturday), E_IotCommunicatorDatatype.type_BOOL);
	ELSIF fbIotWidgets.fbCommand.sVarName = 'stTimeSwitch.stTimeSwitch2.bSunday' THEN
		fbIotWidgets.fbCommand.GetValue(ADR(GVL_Widgets.stWidgetData.stTimeSwitch.stTimeSwitch2.bSunday), SIZEOF(GVL_Widgets.stWidgetData.stTimeSwitch.stTimeSwitch2.bSunday), E_IotCommunicatorDatatype.type_BOOL);
	ELSIF fbIotWidgets.fbCommand.sVarName = 'stTimeSwitch.stTimeSwitch2.tStartTime' THEN
		fbIotWidgets.fbCommand.GetValue(ADR(GVL_Widgets.stWidgetData.stTimeSwitch.stTimeSwitch2.tStartTime), SIZEOF(GVL_Widgets.stWidgetData.stTimeSwitch.stTimeSwitch2.tStartTime), E_IotCommunicatorDatatype.type_TIME_OF_DAY);
	ELSIF fbIotWidgets.fbCommand.sVarName = 'stTimeSwitch.stTimeSwitch2.tEndTime' THEN
		fbIotWidgets.fbCommand.GetValue(ADR(GVL_Widgets.stWidgetData.stTimeSwitch.stTimeSwitch2.tEndTime), SIZEOF(GVL_Widgets.stWidgetData.stTimeSwitch.stTimeSwitch2.tEndTime), E_IotCommunicatorDatatype.type_TIME_OF_DAY);
	//TimeSwitch Sample 3
	ELSIF fbIotWidgets.fbCommand.sVarName = 'stTimeSwitch.stTimeSwitch3.bOn' THEN
		fbIotWidgets.fbCommand.GetValue(ADR(GVL_Widgets.stWidgetData.stTimeSwitch.stTimeSwitch3.bOn), SIZEOF(GVL_Widgets.stWidgetData.stTimeSwitch.stTimeSwitch3.bOn), E_IotCommunicatorDatatype.type_BOOL);
	ELSIF fbIotWidgets.fbCommand.sVarName = 'stTimeSwitch.stTimeSwitch3.bYearly' THEN
		fbIotWidgets.fbCommand.GetValue(ADR(GVL_Widgets.stWidgetData.stTimeSwitch.stTimeSwitch3.bYearly), SIZEOF(GVL_Widgets.stWidgetData.stTimeSwitch.stTimeSwitch3.bYearly), E_IotCommunicatorDatatype.type_BOOL);
	ELSIF fbIotWidgets.fbCommand.sVarName = 'stTimeSwitch.stTimeSwitch3.bMonday' THEN
		fbIotWidgets.fbCommand.GetValue(ADR(GVL_Widgets.stWidgetData.stTimeSwitch.stTimeSwitch3.bMonday), SIZEOF(GVL_Widgets.stWidgetData.stTimeSwitch.stTimeSwitch3.bMonday), E_IotCommunicatorDatatype.type_BOOL);
	ELSIF fbIotWidgets.fbCommand.sVarName = 'stTimeSwitch.stTimeSwitch3.bTuesday' THEN
		fbIotWidgets.fbCommand.GetValue(ADR(GVL_Widgets.stWidgetData.stTimeSwitch.stTimeSwitch3.bTuesday), SIZEOF(GVL_Widgets.stWidgetData.stTimeSwitch.stTimeSwitch3.bTuesday), E_IotCommunicatorDatatype.type_BOOL);
	ELSIF fbIotWidgets.fbCommand.sVarName = 'stTimeSwitch.stTimeSwitch3.bWednesday' THEN
		fbIotWidgets.fbCommand.GetValue(ADR(GVL_Widgets.stWidgetData.stTimeSwitch.stTimeSwitch3.bWednesday), SIZEOF(GVL_Widgets.stWidgetData.stTimeSwitch.stTimeSwitch3.bWednesday), E_IotCommunicatorDatatype.type_BOOL);
	ELSIF fbIotWidgets.fbCommand.sVarName = 'stTimeSwitch.stTimeSwitch3.bThursday' THEN
		fbIotWidgets.fbCommand.GetValue(ADR(GVL_Widgets.stWidgetData.stTimeSwitch.stTimeSwitch3.bThursday), SIZEOF(GVL_Widgets.stWidgetData.stTimeSwitch.stTimeSwitch3.bThursday), E_IotCommunicatorDatatype.type_BOOL);
	ELSIF fbIotWidgets.fbCommand.sVarName = 'stTimeSwitch.stTimeSwitch3.bFriday' THEN
		fbIotWidgets.fbCommand.GetValue(ADR(GVL_Widgets.stWidgetData.stTimeSwitch.stTimeSwitch3.bFriday), SIZEOF(GVL_Widgets.stWidgetData.stTimeSwitch.stTimeSwitch3.bFriday), E_IotCommunicatorDatatype.type_BOOL);
	ELSIF fbIotWidgets.fbCommand.sVarName = 'stTimeSwitch.stTimeSwitch3.bSaturday' THEN
		fbIotWidgets.fbCommand.GetValue(ADR(GVL_Widgets.stWidgetData.stTimeSwitch.stTimeSwitch3.bSaturday), SIZEOF(GVL_Widgets.stWidgetData.stTimeSwitch.stTimeSwitch3.bSaturday), E_IotCommunicatorDatatype.type_BOOL);
	ELSIF fbIotWidgets.fbCommand.sVarName = 'stTimeSwitch.stTimeSwitch3.bSunday' THEN
		fbIotWidgets.fbCommand.GetValue(ADR(GVL_Widgets.stWidgetData.stTimeSwitch.stTimeSwitch3.bSunday), SIZEOF(GVL_Widgets.stWidgetData.stTimeSwitch.stTimeSwitch3.bSunday), E_IotCommunicatorDatatype.type_BOOL);
	ELSIF fbIotWidgets.fbCommand.sVarName = 'stTimeSwitch.stTimeSwitch3.tStartTime' THEN
		fbIotWidgets.fbCommand.GetValue(ADR(GVL_Widgets.stWidgetData.stTimeSwitch.stTimeSwitch3.tStartTime), SIZEOF(GVL_Widgets.stWidgetData.stTimeSwitch.stTimeSwitch3.tStartTime), E_IotCommunicatorDatatype.type_TIME_OF_DAY);
	ELSIF fbIotWidgets.fbCommand.sVarName = 'stTimeSwitch.stTimeSwitch3.tEndTime' THEN
		fbIotWidgets.fbCommand.GetValue(ADR(GVL_Widgets.stWidgetData.stTimeSwitch.stTimeSwitch3.tEndTime), SIZEOF(GVL_Widgets.stWidgetData.stTimeSwitch.stTimeSwitch3.tEndTime), E_IotCommunicatorDatatype.type_TIME_OF_DAY);
	ELSIF fbIotWidgets.fbCommand.sVarName = 'stTimeSwitch.stTimeSwitch3.dStartDate' THEN
		fbIotWidgets.fbCommand.GetValue(ADR(GVL_Widgets.stWidgetData.stTimeSwitch.stTimeSwitch3.dStartDate), SIZEOF(GVL_Widgets.stWidgetData.stTimeSwitch.stTimeSwitch3.dStartDate), E_IotCommunicatorDatatype.type_DATE);
	ELSIF fbIotWidgets.fbCommand.sVarName = 'stTimeSwitch.stTimeSwitch3.dEndDate' THEN
		fbIotWidgets.fbCommand.GetValue(ADR(GVL_Widgets.stWidgetData.stTimeSwitch.stTimeSwitch3.dEndDate), SIZEOF(GVL_Widgets.stWidgetData.stTimeSwitch.stTimeSwitch3.dEndDate), E_IotCommunicatorDatatype.type_DATE);
	ELSIF fbIotWidgets.fbCommand.sVarName = 'stTimeSwitch.stTimeSwitch3.sMode' THEN
		fbIotWidgets.fbCommand.GetValue(ADR(GVL_Widgets.stWidgetData.stTimeSwitch.stTimeSwitch3.sMode), SIZEOF(GVL_Widgets.stWidgetData.stTimeSwitch.stTimeSwitch3.sMode), E_IotCommunicatorDatatype.type_STRING);
	ELSE
		RETURN;
	END_IF
	fbIotWidgets.SendData(ADR(GVL_Widgets.stWidgetData), SIZEOF(GVL_Widgets.stWidgetData));
	fbIotWidgets.fbCommand.Remove();
END_IF
END_METHOD

METHOD ManageVentilation
VAR_INPUT
END_VAR
VAR
END_VAR
//Handling of commands from App
IF fbIotWidgets.fbCommand.bAvailable THEN
	//Ventilation Sample 1 - no processing required - readOnly Widget
	//Ventilation Sample 2 - no mode adjustable, no request value visible
	IF fbIotWidgets.fbCommand.sVarName = 'stVentilation.stVentilation2.bOn' THEN
		fbIotWidgets.fbCommand.GetValue(ADR(GVL_Widgets.stWidgetData.stVentilation.stVentilation2.bOn), SIZEOF(GVL_Widgets.stWidgetData.stVentilation.stVentilation2.bOn), E_IotCommunicatorDatatype.type_BOOL);
	ELSIF fbIotWidgets.fbCommand.sVarName = 'stVentilation.stVentilation2.nValueRequest' THEN
		fbIotWidgets.fbCommand.GetValue(ADR(GVL_Widgets.stWidgetData.stVentilation.stVentilation2.nValueRequest), SIZEOF(GVL_Widgets.stWidgetData.stVentilation.stVentilation2.nValueRequest), E_IotCommunicatorDatatype.type_INT);
	//Ventilation Sample 3
	ELSIF fbIotWidgets.fbCommand.sVarName = 'stVentilation.stVentilation3.bOn' THEN
		fbIotWidgets.fbCommand.GetValue(ADR(GVL_Widgets.stWidgetData.stVentilation.stVentilation3.bOn), SIZEOF(GVL_Widgets.stWidgetData.stVentilation.stVentilation3.bOn), E_IotCommunicatorDatatype.type_BOOL);
	ELSIF fbIotWidgets.fbCommand.sVarName = 'stVentilation.stVentilation3.nValueRequest' THEN
		fbIotWidgets.fbCommand.GetValue(ADR(GVL_Widgets.stWidgetData.stVentilation.stVentilation3.nValueRequest), SIZEOF(GVL_Widgets.stWidgetData.stVentilation.stVentilation3.nValueRequest), E_IotCommunicatorDatatype.type_INT);
	ELSIF fbIotWidgets.fbCommand.sVarName = 'stVentilation.stVentilation3.sMode' THEN
		fbIotWidgets.fbCommand.GetValue(ADR(GVL_Widgets.stWidgetData.stVentilation.stVentilation3.sMode), SIZEOF(GVL_Widgets.stWidgetData.stVentilation.stVentilation3.sMode), E_IotCommunicatorDatatype.type_STRING);
	ELSE
		RETURN;
	END_IF
	fbIotWidgets.SendData(ADR(GVL_Widgets.stWidgetData), SIZEOF(GVL_Widgets.stWidgetData));
	fbIotWidgets.fbCommand.Remove();
END_IF
END_METHOD

METHOD ManageWidgetsOverview
VAR_INPUT
END_VAR
VAR
END_VAR
IF fbIotWidgets.fbCommand.bAvailable THEN
	//Overview Lighting
	IF fbIotWidgets.fbCommand.sVarName = 'stWidgetsOverview.stLighting.bLight' THEN
		fbIotWidgets.fbCommand.GetValue(ADR(GVL_Widgets.stWidgetData.stWidgetsOverview.stLighting.bLight), SIZEOF(GVL_Widgets.stWidgetData.stWidgetsOverview.stLighting.bLight), E_IotCommunicatorDatatype.type_BOOL);
	ELSIF fbIotWidgets.fbCommand.sVarName = 'stWidgetsOverview.stLighting.nLight' THEN
		fbIotWidgets.fbCommand.GetValue(ADR(GVL_Widgets.stWidgetData.stWidgetsOverview.stLighting.nLight), SIZEOF(GVL_Widgets.stWidgetData.stWidgetsOverview.stLighting.nLight), E_IotCommunicatorDatatype.type_INT);
	ELSIF fbIotWidgets.fbCommand.sVarName = 'stWidgetsOverview.stLighting.sMode' THEN
		fbIotWidgets.fbCommand.GetValue(ADR(GVL_Widgets.stWidgetData.stWidgetsOverview.stLighting.sMode), SIZEOF(GVL_Widgets.stWidgetData.stWidgetsOverview.stLighting.sMode), E_IotCommunicatorDatatype.type_STRING);
	//Overview RGBW
	ELSIF fbIotWidgets.fbCommand.sVarName = 'stWidgetsOverview.stRGBW.bLight' THEN
		fbIotWidgets.fbCommand.GetValue(ADR(GVL_Widgets.stWidgetData.stWidgetsOverview.stRGBW.bLight), SIZEOF(GVL_Widgets.stWidgetData.stWidgetsOverview.stRGBW.bLight), E_IotCommunicatorDatatype.type_BOOL);
	ELSIF fbIotWidgets.fbCommand.sVarName = 'stWidgetsOverview.stRGBW.nLight' THEN
		fbIotWidgets.fbCommand.GetValue(ADR(GVL_Widgets.stWidgetData.stWidgetsOverview.stRGBW.nLight), SIZEOF(GVL_Widgets.stWidgetData.stWidgetsOverview.stRGBW.nLight), E_IotCommunicatorDatatype.type_INT);
	ELSIF fbIotWidgets.fbCommand.sVarName = 'stWidgetsOverview.stRGBW.nHueValue' THEN
		fbIotWidgets.fbCommand.GetValue(ADR(GVL_Widgets.stWidgetData.stWidgetsOverview.stRGBW.nHueValue), SIZEOF(GVL_Widgets.stWidgetData.stWidgetsOverview.stRGBW.nHueValue), E_IotCommunicatorDatatype.type_INT);
	ELSIF fbIotWidgets.fbCommand.sVarName = 'stWidgetsOverview.stRGBW.nSaturation' THEN
		fbIotWidgets.fbCommand.GetValue(ADR(GVL_Widgets.stWidgetData.stWidgetsOverview.stRGBW.nSaturation), SIZEOF(GVL_Widgets.stWidgetData.stWidgetsOverview.stRGBW.nSaturation), E_IotCommunicatorDatatype.type_INT);
	ELSIF fbIotWidgets.fbCommand.sVarName = 'stWidgetsOverview.stRGBW.nColorTemperature' THEN
		fbIotWidgets.fbCommand.GetValue(ADR(GVL_Widgets.stWidgetData.stWidgetsOverview.stRGBW.nColorTemperature), SIZEOF(GVL_Widgets.stWidgetData.stWidgetsOverview.stRGBW.nColorTemperature), E_IotCommunicatorDatatype.type_INT);
	ELSIF fbIotWidgets.fbCommand.sVarName = 'stWidgetsOverview.stRGBW.nWhite' THEN
		fbIotWidgets.fbCommand.GetValue(ADR(GVL_Widgets.stWidgetData.stWidgetsOverview.stRGBW.nWhite), SIZEOF(GVL_Widgets.stWidgetData.stWidgetsOverview.stRGBW.nWhite), E_IotCommunicatorDatatype.type_INT);
	ELSIF fbIotWidgets.fbCommand.sVarName = 'stWidgetsOverview.stRGBW.sMode' THEN
		fbIotWidgets.fbCommand.GetValue(ADR(GVL_Widgets.stWidgetData.stWidgetsOverview.stRGBW.sMode), SIZEOF(GVL_Widgets.stWidgetData.stWidgetsOverview.stRGBW.sMode), E_IotCommunicatorDatatype.type_STRING);
	//Overview RGBWEL2564
	ELSIF fbIotWidgets.fbCommand.sVarName = 'stWidgetsOverview.stRGBWLed.bOn' THEN
		fbIotWidgets.fbCommand.GetValue(ADR(GVL_Widgets.stWidgetData.stWidgetsOverview.stRGBWLed.bOn), SIZEOF(GVL_Widgets.stWidgetData.stWidgetsOverview.stRGBWLed.bOn), E_IotCommunicatorDatatype.type_BOOL);
	ELSIF fbIotWidgets.fbCommand.sVarName = 'stWidgetsOverview.stRGBWLed.nGreen' THEN
		fbIotWidgets.fbCommand.GetValue(ADR(GVL_Widgets.stWidgetData.stWidgetsOverview.stRGBWLed.nGreen), SIZEOF(GVL_Widgets.stWidgetData.stWidgetsOverview.stRGBWLed.nGreen), E_IotCommunicatorDatatype.type_INT);
	ELSIF fbIotWidgets.fbCommand.sVarName = 'stWidgetsOverview.stRGBWLed.nBlue' THEN
		fbIotWidgets.fbCommand.GetValue(ADR(GVL_Widgets.stWidgetData.stWidgetsOverview.stRGBWLed.nBlue), SIZEOF(GVL_Widgets.stWidgetData.stWidgetsOverview.stRGBWLed.nBlue), E_IotCommunicatorDatatype.type_INT);
	ELSIF fbIotWidgets.fbCommand.sVarName = 'stWidgetsOverview.stRGBWLed.nRed' THEN
		fbIotWidgets.fbCommand.GetValue(ADR(GVL_Widgets.stWidgetData.stWidgetsOverview.stRGBWLed.nRed), SIZEOF(GVL_Widgets.stWidgetData.stWidgetsOverview.stRGBWLed.nRed), E_IotCommunicatorDatatype.type_INT);
	ELSIF fbIotWidgets.fbCommand.sVarName = 'stWidgetsOverview.stRGBWLed.nWhite' THEN
		fbIotWidgets.fbCommand.GetValue(ADR(GVL_Widgets.stWidgetData.stWidgetsOverview.stRGBWLed.nWhite), SIZEOF(GVL_Widgets.stWidgetData.stWidgetsOverview.stRGBWLed.nWhite), E_IotCommunicatorDatatype.type_INT);
	ELSIF fbIotWidgets.fbCommand.sVarName = 'stWidgetsOverview.stRGBWLed.sMode' THEN
		fbIotWidgets.fbCommand.GetValue(ADR(GVL_Widgets.stWidgetData.stWidgetsOverview.stRGBWLed.sMode), SIZEOF(GVL_Widgets.stWidgetData.stWidgetsOverview.stRGBWLed.sMode), E_IotCommunicatorDatatype.type_STRING);
	//Overview Blinds
	ELSIF fbIotWidgets.fbCommand.sVarName = 'stWidgetsOverview.stBlinds.bPositionUp' THEN
		fbIotWidgets.fbCommand.GetValue(ADR(GVL_Widgets.stWidgetData.stWidgetsOverview.stBlinds.bPositionUp), SIZEOF(GVL_Widgets.stWidgetData.stWidgetsOverview.stBlinds.bPositionUp), E_IotCommunicatorDatatype.type_BOOL);
	ELSIF fbIotWidgets.fbCommand.sVarName = 'stWidgetsOverview.stBlinds.bPositionDown' THEN
		fbIotWidgets.fbCommand.GetValue(ADR(GVL_Widgets.stWidgetData.stWidgetsOverview.stBlinds.bPositionDown), SIZEOF(GVL_Widgets.stWidgetData.stWidgetsOverview.stBlinds.bPositionDown), E_IotCommunicatorDatatype.type_BOOL);
	ELSIF fbIotWidgets.fbCommand.sVarName = 'stWidgetsOverview.stBlinds.nPositionRequest' THEN
		fbIotWidgets.fbCommand.GetValue(ADR(GVL_Widgets.stWidgetData.stWidgetsOverview.stBlinds.nPositionRequest), SIZEOF(GVL_Widgets.stWidgetData.stWidgetsOverview.stBlinds.nPositionRequest), E_IotCommunicatorDatatype.type_INT);
	ELSIF fbIotWidgets.fbCommand.sVarName = 'stWidgetsOverview.stBlinds.bAngleUp' THEN
		fbIotWidgets.fbCommand.GetValue(ADR(GVL_Widgets.stWidgetData.stWidgetsOverview.stBlinds.bAngleUp), SIZEOF(GVL_Widgets.stWidgetData.stWidgetsOverview.stBlinds.bAngleUp), E_IotCommunicatorDatatype.type_BOOL);
	ELSIF fbIotWidgets.fbCommand.sVarName = 'stWidgetsOverview.stBlinds.bAngleDown' THEN
		fbIotWidgets.fbCommand.GetValue(ADR(GVL_Widgets.stWidgetData.stWidgetsOverview.stBlinds.bAngleDown), SIZEOF(GVL_Widgets.stWidgetData.stWidgetsOverview.stBlinds.bAngleDown), E_IotCommunicatorDatatype.type_BOOL);
	ELSIF fbIotWidgets.fbCommand.sVarName = 'stWidgetsOverview.stBlinds.nAngleRequest' THEN
		fbIotWidgets.fbCommand.GetValue(ADR(GVL_Widgets.stWidgetData.stWidgetsOverview.stBlinds.nAngleRequest), SIZEOF(GVL_Widgets.stWidgetData.stWidgetsOverview.stBlinds.nAngleRequest), E_IotCommunicatorDatatype.type_INT);
	ELSIF fbIotWidgets.fbCommand.sVarName = 'stWidgetsOverview.stBlinds.sMode' THEN
		fbIotWidgets.fbCommand.GetValue(ADR(GVL_Widgets.stWidgetData.stWidgetsOverview.stBlinds.sMode), SIZEOF(GVL_Widgets.stWidgetData.stWidgetsOverview.stBlinds.sMode), E_IotCommunicatorDatatype.type_STRING);
	ELSIF fbIotWidgets.fbCommand.sVarName = 'stWidgetsOverview.stBlinds.bActive' THEN
		fbIotWidgets.fbCommand.GetValue(ADR(GVL_Widgets.stWidgetData.stWidgetsOverview.stBlinds.bActive), SIZEOF(GVL_Widgets.stWidgetData.stWidgetsOverview.stBlinds.bActive), E_IotCommunicatorDatatype.type_BOOL);
	//Overview Simple Blinds
	ELSIF fbIotWidgets.fbCommand.sVarName = 'stWidgetsOverview.stSimpleBlinds.bPositionUp' THEN
		fbIotWidgets.fbCommand.GetValue(ADR(GVL_Widgets.stWidgetData.stWidgetsOverview.stSimpleBlinds.bPositionUp), SIZEOF(GVL_Widgets.stWidgetData.stWidgetsOverview.stSimpleBlinds.bPositionUp), E_IotCommunicatorDatatype.type_BOOL);
	ELSIF fbIotWidgets.fbCommand.sVarName = 'stWidgetsOverview.stSimpleBlinds.bPositionDown' THEN
		fbIotWidgets.fbCommand.GetValue(ADR(GVL_Widgets.stWidgetData.stWidgetsOverview.stSimpleBlinds.bPositionDown), SIZEOF(GVL_Widgets.stWidgetData.stWidgetsOverview.stSimpleBlinds.bPositionDown), E_IotCommunicatorDatatype.type_BOOL);
	//Overview Plug
	ELSIF fbIotWidgets.fbCommand.sVarName = 'stWidgetsOverview.stPlug.bOn' THEN
		fbIotWidgets.fbCommand.GetValue(ADR(GVL_Widgets.stWidgetData.stWidgetsOverview.stPlug.bOn), SIZEOF(GVL_Widgets.stWidgetData.stWidgetsOverview.stPlug.bOn), E_IotCommunicatorDatatype.type_BOOL);
	ELSIF fbIotWidgets.fbCommand.sVarName = 'stWidgetsOverview.stPlug.sMode' THEN
		fbIotWidgets.fbCommand.GetValue(ADR(GVL_Widgets.stWidgetData.stWidgetsOverview.stPlug.sMode), SIZEOF(GVL_Widgets.stWidgetData.stWidgetsOverview.stPlug.sMode), E_IotCommunicatorDatatype.type_STRING);
	//Overview AC
	ELSIF fbIotWidgets.fbCommand.sVarName = 'stWidgetsOverview.stAC.nTemperatureRequest' THEN
		fbIotWidgets.fbCommand.GetValue(ADR(GVL_Widgets.stWidgetData.stWidgetsOverview.stAC.nTemperatureRequest), SIZEOF(GVL_Widgets.stWidgetData.stWidgetsOverview.stAC.nTemperatureRequest), E_IotCommunicatorDatatype.type_LREAL);
	ELSIF fbIotWidgets.fbCommand.sVarName = 'stWidgetsOverview.stAC.sMode' THEN
		fbIotWidgets.fbCommand.GetValue(ADR(GVL_Widgets.stWidgetData.stWidgetsOverview.stAC.sMode), SIZEOF(GVL_Widgets.stWidgetData.stWidgetsOverview.stAC.sMode), E_IotCommunicatorDatatype.type_STRING);
	ELSIF fbIotWidgets.fbCommand.sVarName = 'stWidgetsOverview.stAC.sMode_Strength' THEN
		fbIotWidgets.fbCommand.GetValue(ADR(GVL_Widgets.stWidgetData.stWidgetsOverview.stAC.sMode_Strength), SIZEOF(GVL_Widgets.stWidgetData.stWidgetsOverview.stAC.sMode_Strength), E_IotCommunicatorDatatype.type_STRING);
	ELSIF fbIotWidgets.fbCommand.sVarName = 'stWidgetsOverview.stAC.sMode_Lamella' THEN
		fbIotWidgets.fbCommand.GetValue(ADR(GVL_Widgets.stWidgetData.stWidgetsOverview.stAC.sMode_Lamella), SIZEOF(GVL_Widgets.stWidgetData.stWidgetsOverview.stAC.sMode_Lamella), E_IotCommunicatorDatatype.type_STRING);
	//Overview Ventilation
	ELSIF fbIotWidgets.fbCommand.sVarName = 'stWidgetsOverview.stVentilation.bOn' THEN
		fbIotWidgets.fbCommand.GetValue(ADR(GVL_Widgets.stWidgetData.stWidgetsOverview.stVentilation.bOn), SIZEOF(GVL_Widgets.stWidgetData.stWidgetsOverview.stVentilation.bOn), E_IotCommunicatorDatatype.type_BOOL);
	ELSIF fbIotWidgets.fbCommand.sVarName = 'stWidgetsOverview.stVentilation.nValueRequest' THEN
		fbIotWidgets.fbCommand.GetValue(ADR(GVL_Widgets.stWidgetData.stWidgetsOverview.stVentilation.nValueRequest), SIZEOF(GVL_Widgets.stWidgetData.stWidgetsOverview.stVentilation.nValueRequest), E_IotCommunicatorDatatype.type_INT);
	ELSIF fbIotWidgets.fbCommand.sVarName = 'stWidgetsOverview.stVentilation.sMode' THEN
		fbIotWidgets.fbCommand.GetValue(ADR(GVL_Widgets.stWidgetData.stWidgetsOverview.stVentilation.sMode), SIZEOF(GVL_Widgets.stWidgetData.stWidgetsOverview.stVentilation.sMode), E_IotCommunicatorDatatype.type_STRING);
	//Overview Timer Switch
	ELSIF fbIotWidgets.fbCommand.sVarName = 'stWidgetsOverview.stTimeSwitch.bOn' THEN
		fbIotWidgets.fbCommand.GetValue(ADR(GVL_Widgets.stWidgetData.stWidgetsOverview.stTimeSwitch.bOn), SIZEOF(GVL_Widgets.stWidgetData.stWidgetsOverview.stTimeSwitch.bOn), E_IotCommunicatorDatatype.type_BOOL);
	ELSIF fbIotWidgets.fbCommand.sVarName = 'stWidgetsOverview.stTimeSwitch.tStartTime' THEN
		fbIotWidgets.fbCommand.GetValue(ADR(GVL_Widgets.stWidgetData.stWidgetsOverview.stTimeSwitch.tStartTime), SIZEOF(GVL_Widgets.stWidgetData.stWidgetsOverview.stTimeSwitch.tStartTime), E_IotCommunicatorDatatype.type_TIME_OF_DAY);
	ELSIF fbIotWidgets.fbCommand.sVarName = 'stWidgetsOverview.stTimeSwitch.tEndTime' THEN
		fbIotWidgets.fbCommand.GetValue(ADR(GVL_Widgets.stWidgetData.stWidgetsOverview.stTimeSwitch.tEndTime), SIZEOF(GVL_Widgets.stWidgetData.stWidgetsOverview.stTimeSwitch.tEndTime), E_IotCommunicatorDatatype.type_TIME_OF_DAY);
	ELSIF fbIotWidgets.fbCommand.sVarName = 'stWidgetsOverview.stTimeSwitch.dStartDate' THEN
		fbIotWidgets.fbCommand.GetValue(ADR(GVL_Widgets.stWidgetData.stWidgetsOverview.stTimeSwitch.dStartDate), SIZEOF(GVL_Widgets.stWidgetData.stWidgetsOverview.stTimeSwitch.dStartDate), E_IotCommunicatorDatatype.type_DATE);
	ELSIF fbIotWidgets.fbCommand.sVarName = 'stWidgetsOverview.stTimeSwitch.dEndDate' THEN
		fbIotWidgets.fbCommand.GetValue(ADR(GVL_Widgets.stWidgetData.stWidgetsOverview.stTimeSwitch.dEndDate), SIZEOF(GVL_Widgets.stWidgetData.stWidgetsOverview.stTimeSwitch.dEndDate), E_IotCommunicatorDatatype.type_DATE);
	ELSIF fbIotWidgets.fbCommand.sVarName = 'stWidgetsOverview.stTimeSwitch.bYearly' THEN
		fbIotWidgets.fbCommand.GetValue(ADR(GVL_Widgets.stWidgetData.stWidgetsOverview.stTimeSwitch.bYearly), SIZEOF(GVL_Widgets.stWidgetData.stWidgetsOverview.stTimeSwitch.bYearly), E_IotCommunicatorDatatype.type_BOOL);
	ELSIF fbIotWidgets.fbCommand.sVarName = 'stWidgetsOverview.stTimeSwitch.bMonday' THEN
		fbIotWidgets.fbCommand.GetValue(ADR(GVL_Widgets.stWidgetData.stWidgetsOverview.stTimeSwitch.bMonday), SIZEOF(GVL_Widgets.stWidgetData.stWidgetsOverview.stTimeSwitch.bMonday), E_IotCommunicatorDatatype.type_BOOL);
	ELSIF fbIotWidgets.fbCommand.sVarName = 'stWidgetsOverview.stTimeSwitch.bTuesday' THEN
		fbIotWidgets.fbCommand.GetValue(ADR(GVL_Widgets.stWidgetData.stWidgetsOverview.stTimeSwitch.bTuesday), SIZEOF(GVL_Widgets.stWidgetData.stWidgetsOverview.stTimeSwitch.bTuesday), E_IotCommunicatorDatatype.type_BOOL);
	ELSIF fbIotWidgets.fbCommand.sVarName = 'stWidgetsOverview.stTimeSwitch.bWednesday' THEN
		fbIotWidgets.fbCommand.GetValue(ADR(GVL_Widgets.stWidgetData.stWidgetsOverview.stTimeSwitch.bWednesday), SIZEOF(GVL_Widgets.stWidgetData.stWidgetsOverview.stTimeSwitch.bWednesday), E_IotCommunicatorDatatype.type_BOOL);
	ELSIF fbIotWidgets.fbCommand.sVarName = 'stWidgetsOverview.stTimeSwitch.bThursday' THEN
		fbIotWidgets.fbCommand.GetValue(ADR(GVL_Widgets.stWidgetData.stWidgetsOverview.stTimeSwitch.bThursday), SIZEOF(GVL_Widgets.stWidgetData.stWidgetsOverview.stTimeSwitch.bThursday), E_IotCommunicatorDatatype.type_BOOL);
	ELSIF fbIotWidgets.fbCommand.sVarName = 'stWidgetsOverview.stTimeSwitch.bFriday' THEN
		fbIotWidgets.fbCommand.GetValue(ADR(GVL_Widgets.stWidgetData.stWidgetsOverview.stTimeSwitch.bFriday), SIZEOF(GVL_Widgets.stWidgetData.stWidgetsOverview.stTimeSwitch.bFriday), E_IotCommunicatorDatatype.type_BOOL);
	ELSIF fbIotWidgets.fbCommand.sVarName = 'stWidgetsOverview.stTimeSwitch.bSaturday' THEN
		fbIotWidgets.fbCommand.GetValue(ADR(GVL_Widgets.stWidgetData.stWidgetsOverview.stTimeSwitch.bSaturday), SIZEOF(GVL_Widgets.stWidgetData.stWidgetsOverview.stTimeSwitch.bSaturday), E_IotCommunicatorDatatype.type_BOOL);
	ELSIF fbIotWidgets.fbCommand.sVarName = 'stWidgetsOverview.stTimeSwitch.bSunday' THEN
		fbIotWidgets.fbCommand.GetValue(ADR(GVL_Widgets.stWidgetData.stWidgetsOverview.stTimeSwitch.bSunday), SIZEOF(GVL_Widgets.stWidgetData.stWidgetsOverview.stTimeSwitch.bSunday), E_IotCommunicatorDatatype.type_BOOL);
	ELSIF fbIotWidgets.fbCommand.sVarName = 'stWidgetsOverview.stTimeSwitch.sMode' THEN
		fbIotWidgets.fbCommand.GetValue(ADR(GVL_Widgets.stWidgetData.stWidgetsOverview.stTimeSwitch.sMode), SIZEOF(GVL_Widgets.stWidgetData.stWidgetsOverview.stTimeSwitch.sMode), E_IotCommunicatorDatatype.type_STRING);
	//Overview General Widget
	ELSIF fbIotWidgets.fbCommand.sVarName = 'stWidgetsOverview.stGeneral.bValue1' THEN
		fbIotWidgets.fbCommand.GetValue(ADR(GVL_Widgets.stWidgetData.stWidgetsOverview.stGeneral.bValue1), SIZEOF(GVL_Widgets.stWidgetData.stWidgetsOverview.stGeneral.bValue1), E_IotCommunicatorDatatype.type_BOOL);
	ELSIF fbIotWidgets.fbCommand.sVarName = 'stWidgetsOverview.stGeneral.bValue2Up' THEN
		fbIotWidgets.fbCommand.GetValue(ADR(GVL_Widgets.stWidgetData.stWidgetsOverview.stGeneral.bValue2Up), SIZEOF(GVL_Widgets.stWidgetData.stWidgetsOverview.stGeneral.bValue2Up), E_IotCommunicatorDatatype.type_BOOL);
	ELSIF fbIotWidgets.fbCommand.sVarName = 'stWidgetsOverview.stGeneral.bValue2Down' THEN
		fbIotWidgets.fbCommand.GetValue(ADR(GVL_Widgets.stWidgetData.stWidgetsOverview.stGeneral.bValue2Down), SIZEOF(GVL_Widgets.stWidgetData.stWidgetsOverview.stGeneral.bValue2Down), E_IotCommunicatorDatatype.type_BOOL);
	ELSIF fbIotWidgets.fbCommand.sVarName = 'stWidgetsOverview.stGeneral.nValue2Request' THEN
		fbIotWidgets.fbCommand.GetValue(ADR(GVL_Widgets.stWidgetData.stWidgetsOverview.stGeneral.nValue2Request), SIZEOF(GVL_Widgets.stWidgetData.stWidgetsOverview.stGeneral.nValue2Request), E_IotCommunicatorDatatype.type_INT);
	ELSIF fbIotWidgets.fbCommand.sVarName = 'stWidgetsOverview.stGeneral.bValue3Up' THEN
		fbIotWidgets.fbCommand.GetValue(ADR(GVL_Widgets.stWidgetData.stWidgetsOverview.stGeneral.bValue3Up), SIZEOF(GVL_Widgets.stWidgetData.stWidgetsOverview.stGeneral.bValue3Up), E_IotCommunicatorDatatype.type_BOOL);
	ELSIF fbIotWidgets.fbCommand.sVarName = 'stWidgetsOverview.stGeneral.bValue3Down' THEN
		fbIotWidgets.fbCommand.GetValue(ADR(GVL_Widgets.stWidgetData.stWidgetsOverview.stGeneral.bValue3Down), SIZEOF(GVL_Widgets.stWidgetData.stWidgetsOverview.stGeneral.bValue3Down), E_IotCommunicatorDatatype.type_BOOL);
	ELSIF fbIotWidgets.fbCommand.sVarName = 'stWidgetsOverview.stGeneral.nValue3Request' THEN
		fbIotWidgets.fbCommand.GetValue(ADR(GVL_Widgets.stWidgetData.stWidgetsOverview.stGeneral.nValue3Request), SIZEOF(GVL_Widgets.stWidgetData.stWidgetsOverview.stGeneral.nValue3Request), E_IotCommunicatorDatatype.type_INT);
	ELSIF fbIotWidgets.fbCommand.sVarName = 'stWidgetsOverview.stGeneral.sMode1' THEN
		fbIotWidgets.fbCommand.GetValue(ADR(GVL_Widgets.stWidgetData.stWidgetsOverview.stGeneral.sMode1), SIZEOF(GVL_Widgets.stWidgetData.stWidgetsOverview.stGeneral.sMode1), E_IotCommunicatorDatatype.type_STRING);
	ELSIF fbIotWidgets.fbCommand.sVarName = 'stWidgetsOverview.stGeneral.sMode2' THEN
		fbIotWidgets.fbCommand.GetValue(ADR(GVL_Widgets.stWidgetData.stWidgetsOverview.stGeneral.sMode2), SIZEOF(GVL_Widgets.stWidgetData.stWidgetsOverview.stGeneral.sMode2), E_IotCommunicatorDatatype.type_STRING);
	ELSIF fbIotWidgets.fbCommand.sVarName = 'stWidgetsOverview.stGeneral.sMode3' THEN
		fbIotWidgets.fbCommand.GetValue(ADR(GVL_Widgets.stWidgetData.stWidgetsOverview.stGeneral.sMode3), SIZEOF(GVL_Widgets.stWidgetData.stWidgetsOverview.stGeneral.sMode3), E_IotCommunicatorDatatype.type_STRING);
	// Charging Station - Receive Start, Stop, Reserve requests
	ELSIF fbIotWidgets.fbCommand.sVarName = 'stWidgetsOverview.stChargingStation.bStartCharging' THEN
		fbIotWidgets.fbCommand.GetValue(ADR(GVL_Widgets.stWidgetData.stWidgetsOverview.stChargingStation.bStartCharging), SIZEOF(GVL_Widgets.stWidgetData.stWidgetsOverview.stChargingStation.bStartCharging), E_IotCommunicatorDatatype.type_BOOL);
	ELSIF fbIotWidgets.fbCommand.sVarName = 'stWidgetsOverview.stChargingStation.bStopCharging' THEN
		fbIotWidgets.fbCommand.GetValue(ADR(GVL_Widgets.stWidgetData.stWidgetsOverview.stChargingStation.bStopCharging), SIZEOF(GVL_Widgets.stWidgetData.stWidgetsOverview.stChargingStation.bStopCharging), E_IotCommunicatorDatatype.type_BOOL);
	ELSIF fbIotWidgets.fbCommand.sVarName = 'stWidgetsOverview.stChargingStation.bReserveCharging' THEN
		fbIotWidgets.fbCommand.GetValue(ADR(GVL_Widgets.stWidgetData.stWidgetsOverview.stChargingStation.bReserveCharging), SIZEOF(GVL_Widgets.stWidgetData.stWidgetsOverview.stChargingStation.bReserveCharging), E_IotCommunicatorDatatype.type_BOOL);
	ELSE
		RETURN;
	END_IF	
	fbIotWidgets.SendData(ADR(GVL_Widgets.stWidgetData), SIZEOF(GVL_Widgets.stWidgetData));
	fbIotWidgets.fbCommand.Remove();
END_IF
END_METHOD

END_PROGRAM

// ---- POUs/WidgetValues.TcPOU
PROGRAM WidgetValues
VAR
	bInit:BOOL:=TRUE;
	
	aDataSeries			: ARRAY[0..6] OF INT 	:= [850,550,969,1050,1351,255,525];
	aComparismDataSeries: ARRAY[0..6] OF INT 	:= [910,450,950,1234,767,300,175];
	aDataSeriesIdentifier:ARRAY[0..6] OF STRING := ['Mo', 'Di', 'Mi', 'Do', 'Fr', 'Sa', 'So'];
	aLegendLabels		: ARRAY[0..1] OF STRING := ['Week 12 (2024)', 'Week 13 (2024)'];
	
	aMaxPower			: ARRAY[0..2] OF LREAL := [5, 5, 5];
	aCurrentPower		: ARRAY[0..2] OF LREAL := [4.8, 1.2, 2.4];
	aPowerUnits			: ARRAY[0..2] OF STRING := ['W','kW','mW'];
	aAmperage			: ARRAY[0..2] OF LREAL := [10000, 0.0001, 1246387];
	aAmperageCharging	: ARRAY[0..2] OF LREAL := [16, 25, 8];
	aAmperageUnits		: ARRAY[0..2] OF STRING := ['A','A','A'];
	aVoltage			: ARRAY[0..2] OF LREAL := [245120000, 241, 0.000000245];
	aVoltageCharging	: ARRAY[0..2] OF LREAL := [243, 241, 245];
	aVoltageUnits		: ARRAY[0..2] OF STRING := ['V','V','V'];
END_VAR

